	(*Valve 15, A+B*)
	(*Pin #1, 4, 8*)
		Valve15FB
			(
			Enable_Motion:= Enable_Motion,
			Enable_Latch:= TRUE,					(*Enabling Runs Valve as detent type (maintained solenoids*)
			Enable_SideA_PreCharge:= FALSE,		(*Enabling Turns Side A PreCharge Active, reset when Side B is energized in Auto*)
			Enable_SideB_PreCharge:= FALSE,		(*Enabling Turns Side B PreCharge Active, reset when Side A is energized in Auto*)
			PreCharge_Time:= T#0.10S,
			Enable_Auto_Commands:= In_Auto,
			Enable_Manual_Commands:= In_Manual AND (All_Robots_Clear OR TurntableB_At_Robot),  (*TLK ADDED OR*)
			In_Manual_SideA_Command:= (Discrete_In.ManReqs.28 OR Discrete_In.Go_Home),
			In_Manual_SideB_Command:= Discrete_In.ManReqs.29,
			SideA_Indicator:= (Pin1ADVD AND Pin4ADVD AND Pin8ADVD) OR Manual_Ind_HomePrompt,
			SideB_Indicator:= Pin1RETD AND Pin4RETD AND Pin8RETD,
			TurnOn_SideA_SOL=> N100.Q.28,
			TurnOn_SideB_SOL=> N100.Q.29,
			TurnOn_SideA_Indicator=> Manual_Indicators1.28,
			TurnOn_SideB_Indicator=> Manual_Indicators1.29
			 );
		Valve15FB.In_Auto_SideA_Command:= (Clamp_Step.0 AND NOT Unclamp_Step.0 OR Unclamp_Step.3)
										OR ((TurntableA_At_Robot OR Turntable_Bypassed) AND All_Sensors_Off AND Weld_Robots_Clear);
		Valve15FB.In_Auto_SideB_Command:= Unclamp_Step.0;


	(*Valve 16, A+B*)
	(*Clamp #5, 38, Slide #3, 5, 9, 12, 13*)
		Valve16FB
			(
			Enable_Motion:= Enable_Motion,
			Enable_Latch:= TRUE,					(*Enabling Runs Valve as detent type (maintained solenoids*)
			Enable_SideA_PreCharge:= FALSE,		(*Enabling Turns Side A PreCharge Active, reset when Side B is energized in Auto*)
			Enable_SideB_PreCharge:= FALSE,		(*Enabling Turns Side B PreCharge Active, reset when Side A is energized in Auto*)
			PreCharge_Time:= T#0.10S,
			Enable_Auto_Commands:= In_Auto,
			Enable_Manual_Commands:= In_Manual AND (All_Robots_Clear OR TurntableB_At_Robot),  (*TLK ADDED OR*)
			In_Manual_SideA_Command:= Discrete_In.ManReqs.30,
			In_Manual_SideB_Command:= (Discrete_In.ManReqs.31 OR Discrete_In.Go_Home),
			SideA_Indicator:= Clamp5ADVD AND Clamp38ADVD AND Slide3ADVD AND Slide5ADVD AND Slide9ADVD AND Slide12ADVD AND Slide13ADVD,
			SideB_Indicator:= (Clamp5RETD AND Clamp38RETD AND Slide3RETD AND Slide5RETD AND Slide9RETD AND Slide12RETD AND Slide13RETD) OR Manual_Ind_HomePrompt,
			TurnOn_SideA_SOL=> N100.Q.30,
			TurnOn_SideB_SOL=> N100.Q.31,
			TurnOn_SideA_Indicator=> Manual_Indicators1.30,
			TurnOn_SideB_Indicator=> Manual_Indicators1.31
			 );
		Valve16FB.In_Auto_SideA_Command:= (Clamp_Step.4 AND NOT Unclamp_Step.0);
		Valve16FB.In_Auto_SideB_Command:= Unclamp_Step.0
										OR ((TurntableA_At_Robot OR Turntable_Bypassed) AND All_Sensors_Off AND Weld_Robots_Clear);


























(*end*)
END_ACTION

ACTION ValveBank2:


(*+++++++++++THIS AREA IS CUSTOM PER INSTALLATION AND WILL HAVE TO BE MODIFIED PER +++++++++++++*)
(*+++++++++++THIS AREA IS CUSTOM PER INSTALLATION AND WILL HAVE TO BE MODIFIED PER +++++++++++++*)
(*+++++++++++THIS AREA IS CUSTOM PER INSTALLATION AND WILL HAVE TO BE MODIFIED PER +++++++++++++*)

(*+++++++++++VALVE BANK 2 +++++++++++++*)
(*+++++++++++VALVE BANK 2 +++++++++++++*)
(*+++++++++++VALVE BANK 2 +++++++++++++*)


	(*Valve 17, A+B*)
	(*QA Checks #1-6*)
		Valve17FB
			(
			Enable_Motion:= Enable_Motion ,
			Enable_Latch:= TRUE,					(*Enabling Runs Valve as detent type (maintained solenoids*)
			Enable_SideA_PreCharge:= FALSE,		(*Enabling Turns Side A PreCharge Active, reset when Side B is energized in Auto*)
			Enable_SideB_PreCharge:= FALSE,		(*Enabling Turns Side B PreCharge Active, reset when Side A is energized in Auto*)
			PreCharge_Time:= T#0.1S,
			Enable_Auto_Commands:= In_Auto,
			Enable_Manual_Commands:= In_Manual AND (All_Robots_Clear OR TurntableB_At_Robot),  (*TLK ADDED OR*)
			In_Manual_SideA_Command:= Discrete_In.ManReqs2.0,
			In_Manual_SideB_Command:= (Discrete_In.ManReqs2.1 OR Discrete_In.Go_Home),
			SideA_Indicator:= QACheck1ADVD AND QACheck2ADVD AND QACheck3ADVD AND QACheck4ADVD AND QACheck5ADVD AND QACheck6ADVD,
			SideB_Indicator:= (QACheck1RETD AND QACheck2RETD AND QACheck3RETD AND QACheck4RETD AND QACheck5RETD AND QACheck6RETD) OR Manual_Ind_HomePrompt,
			TurnOn_SideA_SOL=> N101.Q.0,
			TurnOn_SideB_SOL=> N101.Q.1,
			TurnOn_SideA_Indicator=> Manual_Indicators2.0,
			TurnOn_SideB_Indicator=> Manual_Indicators2.1
			 );
		Valve17FB.In_Auto_SideA_Command:= CheckQA1FB.Fire_QAchecks AND NOT Cycle_Complete;
		Valve17FB.In_Auto_SideB_Command:= NOT CheckQA1FB.Fire_QAchecks OR (Cycle_Complete AND All_Sensors_Off);


	(*Valve 18, ONLY 543*)
	(*Pin #3, 6*)
		Valve18FB
			(
			Enable_Motion:= Enable_Motion ,
			Enable_Latch:= FALSE,					(*Enabling Runs Valve as detent type (maintained solenoids*)
			Enable_SideA_PreCharge:= FALSE,		(*Enabling Turns Side A PreCharge Active, reset when Side B is energized in Auto*)
			Enable_SideB_PreCharge:= FALSE,		(*Enabling Turns Side B PreCharge Active, reset when Side A is energized in Auto*)
			PreCharge_Time:= T#0.10S,
			Enable_Auto_Commands:= In_Auto,
			Enable_Manual_Commands:= In_Manual AND (All_Robots_Clear OR TurntableB_At_Robot),  (*TLK ADDED OR*)
			In_Manual_SideA_Command:= Discrete_In.ManReqs2.2,
			In_Manual_SideB_Command:= (Discrete_In.ManReqs2.3 OR Discrete_In.Go_Home),
			SideA_Indicator:= Pin3ADVD AND Pin6ADVD,
			SideB_Indicator:= (Pin3RETD AND Pin6RETD) OR Manual_Ind_HomePrompt,
			TurnOn_SideA_SOL=> N101.Q.2,
			TurnOn_SideB_SOL=> N101.Q.3,
			TurnOn_SideA_Indicator=> Manual_Indicators2.2,
			TurnOn_SideB_Indicator=> Manual_Indicators2.3
			 );
	IF ((Model_ID=3) OR (Model_ID=10)) THEN		 
				Valve18FB.In_Auto_SideA_Command:= (Clamp_Step.2 AND NOT Unclamp_Step.0);
				Valve18FB.In_Auto_SideB_Command:= Unclamp_Step.0
												OR ((TurntableA_At_Robot OR Turntable_Bypassed) AND All_Sensors_Off AND Weld_Robots_Clear);
			ELSE
				Valve18FB.In_Auto_SideA_Command:= FALSE;
				Valve18FB.In_Auto_SideB_Command:= TRUE;
			END_IF
												
												
												
	(*Valve 19, ONLY 543*)
	(*Pin #2, 5, 7*)
		Valve19FB
			(
			Enable_Motion:= Enable_Motion,
			Enable_Latch:= FALSE,					(*Enabling Runs Valve as detent type (maintained solenoids*)
			Enable_SideA_PreCharge:= FALSE,		(*Enabling Turns Side A PreCharge Active, reset when Side B is energized in Auto*)
			Enable_SideB_PreCharge:= FALSE,		(*Enabling Turns Side B PreCharge Active, reset when Side A is energized in Auto*)
			PreCharge_Time:= T#0.10S,
			Enable_Auto_Commands:= In_Auto,
			Enable_Manual_Commands:= In_Manual AND (All_Robots_Clear OR TurntableB_At_Robot),  (*TLK ADDED OR*)
			In_Manual_SideA_Command:=  Discrete_In.ManReqs2.4 OR(Discrete_In.Go_Home AND Model_ID=3),
			In_Manual_SideB_Command:=  Discrete_In.ManReqs2.5 OR(Discrete_In.Go_Home AND Model_ID<>3),
			SideA_Indicator:= (Pin2ADVD AND Pin5ADVD AND Pin7ADVD) OR Manual_Ind_HomePrompt,
			SideB_Indicator:= (Pin2RETD AND Pin5RETD AND Pin7RETD) OR Manual_Ind_HomePrompt,
			TurnOn_SideA_SOL=> N101.Q.4,
			TurnOn_SideB_SOL=> N101.Q.5,
			TurnOn_SideA_Indicator=> Manual_Indicators2.4,
			TurnOn_SideB_Indicator=> Manual_Indicators2.5
			 );
	IF ((Model_ID=3) OR (Model_ID=10)) THEN		 
				Valve19FB.In_Auto_SideA_Command:= ((Clamp_Step.0 AND NOT Unclamp_Step.0))
												OR ((TurntableA_At_Robot OR Turntable_Bypassed) AND All_Sensors_Off AND Weld_Robots_Clear);
				Valve19FB.In_Auto_SideB_Command:= Unclamp_Step.0;
		ELSE
				Valve19FB.In_Auto_SideA_Command:= FALSE;
				Valve19FB.In_Auto_SideB_Command:= TRUE;
		END_IF
				
				

	(*Valve 20, ONLY 543*)
	(*Clamp #8, 24, 31*)
		Valve20FB
			(
			Enable_Motion:= Enable_Motion,
			Enable_Latch:= FALSE,					(*Enabling Runs Valve as detent type (maintained solenoids*)
			Enable_SideA_PreCharge:= FALSE,		(*Enabling Turns Side A PreCharge Active, reset when Side B is energized in Auto*)
			Enable_SideB_PreCharge:= FALSE,		(*Enabling Turns Side B PreCharge Active, reset when Side A is energized in Auto*)
			PreCharge_Time:= T#0.10S,
			Enable_Auto_Commands:= In_Auto,
			Enable_Manual_Commands:= In_Manual AND (All_Robots_Clear OR TurntableB_At_Robot),  (*TLK ADDED OR*)
			In_Manual_SideA_Command:= Discrete_In.ManReqs2.6,
			In_Manual_SideB_Command:= (Discrete_In.ManReqs2.7 OR Discrete_In.Go_Home),
			SideA_Indicator:= Clamp8ADVD AND Clamp24ADVD AND Clamp31ADVD,
			SideB_Indicator:= (Clamp8RETD AND Clamp24RETD AND Clamp31RETD) OR Manual_Ind_HomePrompt,
			TurnOn_SideA_SOL=> N101.Q.6,
			TurnOn_SideB_SOL=> N101.Q.7,
			TurnOn_SideA_Indicator=> Manual_Indicators2.6,
			TurnOn_SideB_Indicator=> Manual_Indicators2.7
			 );
			 
	IF ((Model_ID=3) OR (Model_ID=10)) THEN			 
				Valve20FB.In_Auto_SideA_Command:= (Clamp_Step.1 AND NOT Unclamp_Step.3);
				Valve20FB.In_Auto_SideB_Command:= Unclamp_Step.3
												OR ((TurntableA_At_Robot OR Turntable_Bypassed) AND All_Sensors_Off AND Weld_Robots_Clear);
		ELSE
				Valve20FB.In_Auto_SideA_Command:= FALSE;
				Valve20FB.In_Auto_SideB_Command:= TRUE;
		END_IF


	(*Valve 21, ONLY 543*)
	(*Clamp #10, 27*)
		Valve21FB
			(
			Enable_Motion:= Enable_Motion,
			Enable_Latch:= FALSE,					(*Enabling Runs Valve as detent type (maintained solenoids*)
			Enable_SideA_PreCharge:= FALSE,		(*Enabling Turns Side A PreCharge Active, reset when Side B is energized in Auto*)
			Enable_SideB_PreCharge:= FALSE,		(*Enabling Turns Side B PreCharge Active, reset when Side A is energized in Auto*)
			PreCharge_Time:= T#0.10S,
			Enable_Auto_Commands:= In_Auto,
			Enable_Manual_Commands:= In_Manual AND (All_Robots_Clear OR TurntableB_At_Robot),  (*TLK ADDED OR*)
			In_Manual_SideA_Command:= Discrete_In.ManReqs2.8,
			In_Manual_SideB_Command:= (Discrete_In.ManReqs2.9 OR Discrete_In.Go_Home),
			SideA_Indicator:= Clamp10ADVD AND Clamp27ADVD,
			SideB_Indicator:= (Clamp10RETD AND Clamp27RETD) OR Manual_Ind_HomePrompt,
			TurnOn_SideA_SOL=> N101.Q.8,
			TurnOn_SideB_SOL=> N101.Q.9,
			TurnOn_SideA_Indicator=> Manual_Indicators2.8,
			TurnOn_SideB_Indicator=> Manual_Indicators2.9
			 );
	IF ((Model_ID=3) OR (Model_ID=10)) THEN			 
				Valve21FB.In_Auto_SideA_Command:= (Clamp_Step.1 AND NOT Unclamp_Step.3);
				Valve21FB.In_Auto_SideB_Command:= Unclamp_Step.3
												OR ((TurntableA_At_Robot OR Turntable_Bypassed) AND All_Sensors_Off AND Weld_Robots_Clear);
		ELSE
				Valve21FB.In_Auto_SideA_Command:= FALSE;
				Valve21FB.In_Auto_SideB_Command:= TRUE;
		END_IF

	(*Valve 22, A+B*)
	(*LOCKS*)
		Valve22FB
			(
			Enable_Motion:= Enable_Motion ,
			Enable_Latch:= FALSE,					(*Enabling Runs Valve as detent type (maintained solenoids*)
			Enable_SideA_PreCharge:= FALSE,		(*Enabling Turns Side A PreCharge Active, reset when Side B is energized in Auto*)
			Enable_SideB_PreCharge:= FALSE,		(*Enabling Turns Side B PreCharge Active, reset when Side A is energized in Auto*)
			PreCharge_Time:= T#0.10S,
			Enable_Auto_Commands:= In_Auto,
			Enable_Manual_Commands:= In_Manual AND (All_Robots_Clear OR TurntableB_At_Robot),  (*TLK ADDED OR*)
			In_Manual_SideA_Command:= (Discrete_In.ManReqs2.10 OR Discrete_In.Go_Home)
										OR (N100.Q.18 AND NOT (Slide4ADVD AND Slide8ADVD AND Slide11ADVD))
										OR (N100.Q.19 AND NOT (Slide4RETD AND Slide8RETD AND Slide11RETD))
										OR (N100.Q.20 AND NOT (Slide6ADVD))
										OR (N100.Q.21 AND NOT (Slide6RETD))
										OR (N100.Q.22 AND NOT (Slide7ADVD))
										OR (N100.Q.23 AND NOT (Slide7RETD))
										OR (N100.Q.24 AND NOT (Slide10ADVD))
										OR (N100.Q.25 AND NOT (Slide10RETD))
										OR (N100.Q.26 AND NOT (Slide1ADVD AND Slide2ADVD AND Slide14ADVD AND Slide15ADVD))
										OR (N100.Q.27 AND NOT (Slide1RETD AND Slide2RETD AND Slide14RETD AND Slide15RETD))
										OR (N100.Q.30 AND NOT (Slide3ADVD AND Slide5ADVD AND Slide9ADVD AND Slide12ADVD AND Slide13ADVD))
										OR (N100.Q.31 AND NOT (Slide3RETD AND Slide5RETD AND Slide9RETD AND Slide12RETD AND Slide13RETD)),
			In_Manual_SideB_Command:= FALSE,
			SideA_Indicator:= Manual_Ind_HomePrompt,
			SideB_Indicator:= FALSE,
			TurnOn_SideA_SOL=> N101.Q.10,
			TurnOn_SideB_SOL=> N101.Q.11,
			TurnOn_SideA_Indicator=> Manual_Indicators2.10,
			TurnOn_SideB_Indicator=> Manual_Indicators2.11
			 );
		Valve22FB.In_Auto_SideA_Command:= (N100.Q.18 AND NOT (Slide4ADVD AND Slide8ADVD AND Slide11ADVD))
										OR (N100.Q.19 AND NOT (Slide4RETD AND Slide8RETD AND Slide11RETD))
										OR (N100.Q.20 AND NOT (Slide6ADVD))
										OR (N100.Q.21 AND NOT (Slide6RETD))
										OR (N100.Q.22 AND NOT (Slide7ADVD))
										OR (N100.Q.23 AND NOT (Slide7RETD))
										OR (N100.Q.24 AND NOT (Slide10ADVD))
										OR (N100.Q.25 AND NOT (Slide10RETD))
										OR (N100.Q.26 AND NOT (Slide1ADVD AND Slide2ADVD AND Slide14ADVD AND Slide15ADVD))
										OR (N100.Q.27 AND NOT (Slide1RETD AND Slide2RETD AND Slide14RETD AND Slide15RETD))
										OR (N100.Q.30 AND NOT (Slide3ADVD AND Slide5ADVD AND Slide9ADVD AND Slide12ADVD AND Slide13ADVD))
										OR (N100.Q.31 AND NOT (Slide3RETD AND Slide5RETD AND Slide9RETD AND Slide12RETD AND Slide13RETD));
		Valve22FB.In_Auto_SideB_Command:= FALSE;

	(*Valve 23, A+B*)
	(*Spare*)
		Valve23FB
			(
			Enable_Motion:= Enable_Motion,
			Enable_Latch:= FALSE,					(*Enabling Runs Valve as detent type (maintained solenoids*)
			Enable_SideA_PreCharge:= FALSE,		(*Enabling Turns Side A PreCharge Active, reset when Side B is energized in Auto*)
			Enable_SideB_PreCharge:= FALSE,		(*Enabling Turns Side B PreCharge Active, reset when Side A is energized in Auto*)
			PreCharge_Time:= T#0.10S,
			Enable_Auto_Commands:= In_Auto,
			Enable_Manual_Commands:= In_Manual AND (All_Robots_Clear OR TurntableB_At_Robot),  (*TLK ADDED OR*)
			In_Manual_SideA_Command:= Discrete_In.ManReqs2.12,
			In_Manual_SideB_Command:= Discrete_In.ManReqs2.13 OR Discrete_In.Go_Home,
			SideA_Indicator:= (*Clamp21ADVD*) FALSE,
			SideB_Indicator:= (*Clamp21RETD*) FALSE,
			TurnOn_SideA_SOL=> N101.Q.12,
			TurnOn_SideB_SOL=> N101.Q.13,
			TurnOn_SideA_Indicator=> Manual_Indicators2.12,
			TurnOn_SideB_Indicator=> Manual_Indicators2.13
			 );
		Valve23FB.In_Auto_SideA_Command:= (*Clamp_Step.1 AND NOT Unclamp_Step.0*) FALSE;
		Valve23FB.In_Auto_SideB_Command:= (*Unclamp_Step.0
										OR ((TurntableA_At_Robot OR Turntable_Bypassed) AND All_Sensors_Off AND Weld_Robots_Clear)*) FALSE;


(*---------------------------------------------------------SPARE---------------------------------------------------------*)		


	(*Valve 24, A+B*)
	(*spare*)
		Valve24FB
			(
			Enable_Motion:= Enable_Motion ,
			Enable_Latch:= TRUE,					(*Enabling Runs Valve as detent type (maintained solenoids*)
			Enable_SideA_PreCharge:= FALSE,		(*Enabling Turns Side A PreCharge Active, reset when Side B is energized in Auto*)
			Enable_SideB_PreCharge:= FALSE,		(*Enabling Turns Side B PreCharge Active, reset when Side A is energized in Auto*)
			PreCharge_Time:= T#0.10S,
			Enable_Auto_Commands:= In_Auto,
			Enable_Manual_Commands:= In_Manual AND (All_Robots_Clear OR TurntableB_At_Robot),  (*TLK ADDED OR*)
			In_Manual_SideA_Command:= Discrete_In.ManReqs2.14,
			In_Manual_SideB_Command:= Discrete_In.ManReqs2.15,
			SideA_Indicator:= FALSE,
			SideB_Indicator:= FALSE,
			TurnOn_SideA_SOL=> N101.Q.14,
			TurnOn_SideB_SOL=> N101.Q.15,
			TurnOn_SideA_Indicator=> Manual_Indicators2.14,
			TurnOn_SideB_Indicator=> Manual_Indicators2.15
			 );
		Valve24FB.In_Auto_SideA_Command:= FALSE;
		Valve24FB.In_Auto_SideB_Command:= FALSE;


	(*Valve 25, A+B*)
	(*spare*)
		Valve25FB
			(
			Enable_Motion:= Enable_Motion ,
			Enable_Latch:= TRUE,					(*Enabling Runs Valve as detent type (maintained solenoids*)
			Enable_SideA_PreCharge:= FALSE,		(*Enabling Turns Side A PreCharge Active, reset when Side B is energized in Auto*)
			Enable_SideB_PreCharge:= FALSE,		(*Enabling Turns Side B PreCharge Active, reset when Side A is energized in Auto*)
			PreCharge_Time:= T#0.10S,
			Enable_Auto_Commands:= In_Auto,
			Enable_Manual_Commands:= In_Manual AND (All_Robots_Clear OR TurntableB_At_Robot),  (*TLK ADDED OR*)
			In_Manual_SideA_Command:= Discrete_In.ManReqs2.16,
			In_Manual_SideB_Command:= Discrete_In.ManReqs2.17,
			SideA_Indicator:= FALSE,
			SideB_Indicator:= FALSE,
			TurnOn_SideA_SOL=> N101.Q.16,
			TurnOn_SideB_SOL=> N101.Q.17,
			TurnOn_SideA_Indicator=> Manual_Indicators2.16,
			TurnOn_SideB_Indicator=> Manual_Indicators2.17
			 );
		Valve25FB.In_Auto_SideA_Command:= FALSE;
		Valve25FB.In_Auto_SideB_Command:= FALSE;


	(*Valve 26, A+B*)
	(*spare*)
		Valve26FB
			(
			Enable_Motion:= Enable_Motion ,
			Enable_Latch:= TRUE,					(*Enabling Runs Valve as detent type (maintained solenoids*)
			Enable_SideA_PreCharge:= FALSE,		(*Enabling Turns Side A PreCharge Active, reset when Side B is energized in Auto*)
			Enable_SideB_PreCharge:= FALSE,		(*Enabling Turns Side B PreCharge Active, reset when Side A is energized in Auto*)
			PreCharge_Time:= T#0.10S,
			Enable_Auto_Commands:= In_Auto,
			Enable_Manual_Commands:= In_Manual AND (All_Robots_Clear OR TurntableB_At_Robot),  (*TLK ADDED OR*)
			In_Manual_SideA_Command:= Discrete_In.ManReqs2.18,
			In_Manual_SideB_Command:= Discrete_In.ManReqs2.19,
			SideA_Indicator:= FALSE,
			SideB_Indicator:= FALSE,
			TurnOn_SideA_SOL=> N101.Q.18,
			TurnOn_SideB_SOL=> N101.Q.19,
			TurnOn_SideA_Indicator=> Manual_Indicators2.18,
			TurnOn_SideB_Indicator=> Manual_Indicators2.19
			 );
		Valve26FB.In_Auto_SideA_Command:= FALSE;
		Valve26FB.In_Auto_SideB_Command:= FALSE;


	(*Valve 27, A+B*)
	(*spare*)
		Valve27FB
			(
			Enable_Motion:= Enable_Motion ,
			Enable_Latch:= TRUE,					(*Enabling Runs Valve as detent type (maintained solenoids*)
			Enable_SideA_PreCharge:= FALSE,		(*Enabling Turns Side A PreCharge Active, reset when Side B is energized in Auto*)
			Enable_SideB_PreCharge:= FALSE,		(*Enabling Turns Side B PreCharge Active, reset when Side A is energized in Auto*)
			PreCharge_Time:= T#0.10S,
			Enable_Auto_Commands:= In_Auto,
			Enable_Manual_Commands:= In_Manual AND (All_Robots_Clear OR TurntableB_At_Robot),  (*TLK ADDED OR*)
			In_Manual_SideA_Command:= Discrete_In.ManReqs2.20,
			In_Manual_SideB_Command:= Discrete_In.ManReqs2.21,
			SideA_Indicator:= FALSE,
			SideB_Indicator:= FALSE,
			TurnOn_SideA_SOL=> N101.Q.20,
			TurnOn_SideB_SOL=> N101.Q.21,
			TurnOn_SideA_Indicator=> Manual_Indicators2.20,
			TurnOn_SideB_Indicator=> Manual_Indicators2.21
			 );
		Valve27FB.In_Auto_SideA_Command:= FALSE;
		Valve27FB.In_Auto_SideB_Command:= FALSE;


	(*Valve 28, A+B*)
	(*spare*)
		Valve28FB
			(
			Enable_Motion:= Enable_Motion ,
			Enable_Latch:= TRUE,					(*Enabling Runs Valve as detent type (maintained solenoids*)
			Enable_SideA_PreCharge:= FALSE,		(*Enabling Turns Side A PreCharge Active, reset when Side B is energized in Auto*)
			Enable_SideB_PreCharge:= FALSE,		(*Enabling Turns Side B PreCharge Active, reset when Side A is energized in Auto*)
			PreCharge_Time:= T#0.10S,
			Enable_Auto_Commands:= In_Auto,
			Enable_Manual_Commands:= In_Manual AND (All_Robots_Clear OR TurntableB_At_Robot),  (*TLK ADDED OR*)
			In_Manual_SideA_Command:= Discrete_In.ManReqs2.22,
			In_Manual_SideB_Command:= Discrete_In.ManReqs2.23,
			SideA_Indicator:= FALSE,
			SideB_Indicator:= FALSE,
			TurnOn_SideA_SOL=> N101.Q.22,
			TurnOn_SideB_SOL=> N101.Q.23,
			TurnOn_SideA_Indicator=> Manual_Indicators2.22,
			TurnOn_SideB_Indicator=> Manual_Indicators2.23
			 );
		Valve28FB.In_Auto_SideA_Command:= FALSE;
		Valve28FB.In_Auto_SideB_Command:= FALSE;


	(*Valve 29, A+B*)
	(*spare*)
		Valve29FB
			(
			Enable_Motion:= Enable_Motion ,
			Enable_Latch:= TRUE,					(*Enabling Runs Valve as detent type (maintained solenoids*)
			Enable_SideA_PreCharge:= FALSE,		(*Enabling Turns Side A PreCharge Active, reset when Side B is energized in Auto*)
			Enable_SideB_PreCharge:= FALSE,		(*Enabling Turns Side B PreCharge Active, reset when Side A is energized in Auto*)
			PreCharge_Time:= T#0.10S,
			Enable_Auto_Commands:= In_Auto,
			Enable_Manual_Commands:= In_Manual AND (All_Robots_Clear OR TurntableB_At_Robot),  (*TLK ADDED OR*)
			In_Manual_SideA_Command:= Discrete_In.ManReqs2.24,
			In_Manual_SideB_Command:= Discrete_In.ManReqs2.25,
			SideA_Indicator:= FALSE,
			SideB_Indicator:= FALSE,
			TurnOn_SideA_SOL=> N101.Q.24,
			TurnOn_SideB_SOL=> N101.Q.25,
			TurnOn_SideA_Indicator=> Manual_Indicators2.24,
			TurnOn_SideB_Indicator=> Manual_Indicators2.25
			 );
		Valve29FB.In_Auto_SideA_Command:= FALSE;
		Valve29FB.In_Auto_SideB_Command:= FALSE;


	(*Valve 30, A+B*)
	(*spare*)
		Valve30FB
			(
			Enable_Motion:= Enable_Motion ,
			Enable_Latch:= TRUE,					(*Enabling Runs Valve as detent type (maintained solenoids*)
			Enable_SideA_PreCharge:= FALSE,		(*Enabling Turns Side A PreCharge Active, reset when Side B is energized in Auto*)
			Enable_SideB_PreCharge:= FALSE,		(*Enabling Turns Side B PreCharge Active, reset when Side A is energized in Auto*)
			PreCharge_Time:= T#0.10S,
			Enable_Auto_Commands:= In_Auto,
			Enable_Manual_Commands:= In_Manual AND (All_Robots_Clear OR TurntableB_At_Robot),  (*TLK ADDED OR*)
			In_Manual_SideA_Command:= Discrete_In.ManReqs2.26,
			In_Manual_SideB_Command:= Discrete_In.ManReqs2.27,
			SideA_Indicator:= FALSE,
			SideB_Indicator:= FALSE,
			TurnOn_SideA_SOL=> N101.Q.26,
			TurnOn_SideB_SOL=> N101.Q.27,
			TurnOn_SideA_Indicator=> Manual_Indicators2.26,
			TurnOn_SideB_Indicator=> Manual_Indicators2.27
			 );
		Valve30FB.In_Auto_SideA_Command:= FALSE;
		Valve30FB.In_Auto_SideB_Command:= FALSE;


	(*Valve 31, A+B*)
	(*spare*)
		Valve31FB
			(
			Enable_Motion:= Enable_Motion ,
			Enable_Latch:= TRUE,					(*Enabling Runs Valve as detent type (maintained solenoids*)
			Enable_SideA_PreCharge:= FALSE,		(*Enabling Turns Side A PreCharge Active, reset when Side B is energized in Auto*)
			Enable_SideB_PreCharge:= FALSE,		(*Enabling Turns Side B PreCharge Active, reset when Side A is energized in Auto*)
			PreCharge_Time:= T#0.10S,
			Enable_Auto_Commands:= In_Auto,
			Enable_Manual_Commands:= In_Manual AND (All_Robots_Clear OR TurntableB_At_Robot),  (*TLK ADDED OR*)
			In_Manual_SideA_Command:= Discrete_In.ManReqs2.28,
			In_Manual_SideB_Command:= Discrete_In.ManReqs2.29,
			SideA_Indicator:= FALSE,
			SideB_Indicator:= FALSE,
			TurnOn_SideA_SOL=> N101.Q.28,
			TurnOn_SideB_SOL=> N101.Q.29,
			TurnOn_SideA_Indicator=> Manual_Indicators2.28,
			TurnOn_SideB_Indicator=> Manual_Indicators2.29
			 );
		Valve31FB.In_Auto_SideA_Command:= FALSE;
		Valve31FB.In_Auto_SideB_Command:= FALSE;


	(*Valve 32, A+B*)
	(*spare*)
		Valve32FB
			(
			Enable_Motion:= Enable_Motion ,
			Enable_Latch:= TRUE,					(*Enabling Runs Valve as detent type (maintained solenoids*)
			Enable_SideA_PreCharge:= FALSE,		(*Enabling Turns Side A PreCharge Active, reset when Side B is energized in Auto*)
			Enable_SideB_PreCharge:= FALSE,		(*Enabling Turns Side B PreCharge Active, reset when Side A is energized in Auto*)
			PreCharge_Time:= T#0.10S,
			Enable_Auto_Commands:= In_Auto,
			Enable_Manual_Commands:= In_Manual AND (All_Robots_Clear OR TurntableB_At_Robot),  (*TLK ADDED OR*)
			In_Manual_SideA_Command:= Discrete_In.ManReqs2.30,
			In_Manual_SideB_Command:= Discrete_In.ManReqs2.31,
			SideA_Indicator:= FALSE,
			SideB_Indicator:= FALSE,
			TurnOn_SideA_SOL=> N101.Q.30,
			TurnOn_SideB_SOL=> N101.Q.31,
			TurnOn_SideA_Indicator=> Manual_Indicators2.30,
			TurnOn_SideB_Indicator=> Manual_Indicators2.31
			 );
		Valve32FB.In_Auto_SideA_Command:= FALSE;
		Valve32FB.In_Auto_SideB_Command:= FALSE;




















(*end*)
END_ACTION

ACTION ValveBank3:


(*+++++++++++THIS AREA IS CUSTOM PER INSTALLATION AND WILL HAVE TO BE MODIFIED PER +++++++++++++*)
(*+++++++++++THIS AREA IS CUSTOM PER INSTALLATION AND WILL HAVE TO BE MODIFIED PER +++++++++++++*)
(*+++++++++++THIS AREA IS CUSTOM PER INSTALLATION AND WILL HAVE TO BE MODIFIED PER +++++++++++++*)

(*+++++++++++VALVE BANK 3 +++++++++++++*)
(*+++++++++++VALVE BANK 3 +++++++++++++*)
(*+++++++++++VALVE BANK 3 +++++++++++++*)


	(*Valve 33, A+B*)
	(*spare*)
		Valve33FB
			(
			Enable_Motion:= Enable_Motion ,
			Enable_Latch:= TRUE,					(*Enabling Runs Valve as detent type (maintained solenoids*)
			Enable_SideA_PreCharge:= FALSE,		(*Enabling Turns Side A PreCharge Active, reset when Side B is energized in Auto*)
			Enable_SideB_PreCharge:= FALSE,		(*Enabling Turns Side B PreCharge Active, reset when Side A is energized in Auto*)
			PreCharge_Time:= T#0.1S,
			Enable_Auto_Commands:= In_Auto,
			Enable_Manual_Commands:= In_Manual AND All_Robots_Clear,
			In_Manual_SideA_Command:= Discrete_In.ManReqs3.0,
			In_Manual_SideB_Command:= (Discrete_In.ManReqs3.1 OR Discrete_In.Go_Home),
			SideA_Indicator:= FALSE,
			SideB_Indicator:= FALSE,
			TurnOn_SideA_SOL=> N102.Q.0,
			TurnOn_SideB_SOL=> N102.Q.1,
			TurnOn_SideA_Indicator=> Manual_Indicators3.0,
			TurnOn_SideB_Indicator=> Manual_Indicators3.1
			 );
		Valve33FB.In_Auto_SideA_Command:= FALSE;
		Valve33FB.In_Auto_SideB_Command:= FALSE;


	(*Valve 34, A+B*)
	(*spare*)
		Valve34FB
			(
			Enable_Motion:= Enable_Motion ,
			Enable_Latch:= TRUE,					(*Enabling Runs Valve as detent type (maintained solenoids*)
			Enable_SideA_PreCharge:= FALSE,		(*Enabling Turns Side A PreCharge Active, reset when Side B is energized in Auto*)
			Enable_SideB_PreCharge:= FALSE,		(*Enabling Turns Side B PreCharge Active, reset when Side A is energized in Auto*)
			PreCharge_Time:= T#0.10S,
			Enable_Auto_Commands:= In_Auto,
			Enable_Manual_Commands:= In_Manual AND All_Robots_Clear,
			In_Manual_SideA_Command:= Discrete_In.ManReqs3.2,
			In_Manual_SideB_Command:= Discrete_In.ManReqs3.3,
			SideA_Indicator:= FALSE,
			SideB_Indicator:= FALSE,
			TurnOn_SideA_SOL=> N102.Q.2,
			TurnOn_SideB_SOL=> N102.Q.3,
			TurnOn_SideA_Indicator=> Manual_Indicators3.2,
			TurnOn_SideB_Indicator=> Manual_Indicators3.3
			 );
		Valve34FB.In_Auto_SideA_Command:= FALSE;
		Valve34FB.In_Auto_SideB_Command:= FALSE;


	(*Valve 35, A+B*)
	(*spare*)
		Valve35FB
			(
			Enable_Motion:= Enable_Motion ,
			Enable_Latch:= TRUE,					(*Enabling Runs Valve as detent type (maintained solenoids*)
			Enable_SideA_PreCharge:= FALSE,		(*Enabling Turns Side A PreCharge Active, reset when Side B is energized in Auto*)
			Enable_SideB_PreCharge:= FALSE,		(*Enabling Turns Side B PreCharge Active, reset when Side A is energized in Auto*)
			PreCharge_Time:= T#0.10S,
			Enable_Auto_Commands:= In_Auto,
			Enable_Manual_Commands:= In_Manual AND All_Robots_Clear,
			In_Manual_SideA_Command:= Discrete_In.ManReqs3.4,
			In_Manual_SideB_Command:= Discrete_In.ManReqs3.5,
			SideA_Indicator:= FALSE,
			SideB_Indicator:= FALSE,
			TurnOn_SideA_SOL=> N102.Q.4,
			TurnOn_SideB_SOL=> N102.Q.5,
			TurnOn_SideA_Indicator=> Manual_Indicators3.4,
			TurnOn_SideB_Indicator=> Manual_Indicators3.5
			 );
		Valve35FB.In_Auto_SideA_Command:= FALSE;
		Valve35FB.In_Auto_SideB_Command:= FALSE;


	(*Valve 36, A+B*)
	(*spare*)
		Valve36FB
			(
			Enable_Motion:= Enable_Motion ,
			Enable_Latch:= TRUE,					(*Enabling Runs Valve as detent type (maintained solenoids*)
			Enable_SideA_PreCharge:= FALSE,		(*Enabling Turns Side A PreCharge Active, reset when Side B is energized in Auto*)
			Enable_SideB_PreCharge:= FALSE,		(*Enabling Turns Side B PreCharge Active, reset when Side A is energized in Auto*)
			PreCharge_Time:= T#0.10S,
			Enable_Auto_Commands:= In_Auto,
			Enable_Manual_Commands:= In_Manual AND All_Robots_Clear,
			In_Manual_SideA_Command:= Discrete_In.ManReqs3.6,
			In_Manual_SideB_Command:= Discrete_In.ManReqs3.7,
			SideA_Indicator:= FALSE,
			SideB_Indicator:= FALSE,
			TurnOn_SideA_SOL=> N102.Q.6,
			TurnOn_SideB_SOL=> N102.Q.7,
			TurnOn_SideA_Indicator=> Manual_Indicators3.6,
			TurnOn_SideB_Indicator=> Manual_Indicators3.7
			 );
		Valve36FB.In_Auto_SideA_Command:= FALSE;
		Valve36FB.In_Auto_SideB_Command:= FALSE;


	(*Valve 37, A+B*)
	(*spare*)
		Valve37FB
			(
			Enable_Motion:= Enable_Motion ,
			Enable_Latch:= TRUE,					(*Enabling Runs Valve as detent type (maintained solenoids*)
			Enable_SideA_PreCharge:= FALSE,		(*Enabling Turns Side A PreCharge Active, reset when Side B is energized in Auto*)
			Enable_SideB_PreCharge:= FALSE,		(*Enabling Turns Side B PreCharge Active, reset when Side A is energized in Auto*)
			PreCharge_Time:= T#0.10S,
			Enable_Auto_Commands:= In_Auto,
			Enable_Manual_Commands:= In_Manual AND All_Robots_Clear,
			In_Manual_SideA_Command:= Discrete_In.ManReqs3.8,
			In_Manual_SideB_Command:= Discrete_In.ManReqs3.9,
			SideA_Indicator:= FALSE,
			SideB_Indicator:= FALSE,
			TurnOn_SideA_SOL=> N102.Q.8,
			TurnOn_SideB_SOL=> N102.Q.9,
			TurnOn_SideA_Indicator=> Manual_Indicators3.8,
			TurnOn_SideB_Indicator=> Manual_Indicators3.9
			 );
		Valve37FB.In_Auto_SideA_Command:= FALSE;
		Valve37FB.In_Auto_SideB_Command:= FALSE;


	(*Valve 38, A+B*)
	(*spare*)
		Valve38FB
			(
			Enable_Motion:= Enable_Motion ,
			Enable_Latch:= TRUE,					(*Enabling Runs Valve as detent type (maintained solenoids*)
			Enable_SideA_PreCharge:= FALSE,		(*Enabling Turns Side A PreCharge Active, reset when Side B is energized in Auto*)
			Enable_SideB_PreCharge:= FALSE,		(*Enabling Turns Side B PreCharge Active, reset when Side A is energized in Auto*)
			PreCharge_Time:= T#0.10S,
			Enable_Auto_Commands:= In_Auto,
			Enable_Manual_Commands:= In_Manual AND All_Robots_Clear,
			In_Manual_SideA_Command:= Discrete_In.ManReqs3.10,
			In_Manual_SideB_Command:= Discrete_In.ManReqs3.11,
			SideA_Indicator:= FALSE,
			SideB_Indicator:= FALSE,
			TurnOn_SideA_SOL=> N102.Q.10,
			TurnOn_SideB_SOL=> N102.Q.11,
			TurnOn_SideA_Indicator=> Manual_Indicators3.10,
			TurnOn_SideB_Indicator=> Manual_Indicators3.11
			 );
		Valve38FB.In_Auto_SideA_Command:= FALSE;
		Valve38FB.In_Auto_SideB_Command:= FALSE;


	(*Valve 39, A+B*)
	(*spare*)
		Valve39FB
			(
			Enable_Motion:= Enable_Motion ,
			Enable_Latch:= TRUE,					(*Enabling Runs Valve as detent type (maintained solenoids*)
			Enable_SideA_PreCharge:= FALSE,		(*Enabling Turns Side A PreCharge Active, reset when Side B is energized in Auto*)
			Enable_SideB_PreCharge:= FALSE,		(*Enabling Turns Side B PreCharge Active, reset when Side A is energized in Auto*)
			PreCharge_Time:= T#0.10S,
			Enable_Auto_Commands:= In_Auto,
			Enable_Manual_Commands:= In_Manual AND All_Robots_Clear,
			In_Manual_SideA_Command:= Discrete_In.ManReqs3.12,
			In_Manual_SideB_Command:= Discrete_In.ManReqs3.13,
			SideA_Indicator:= FALSE,
			SideB_Indicator:= FALSE,
			TurnOn_SideA_SOL=> N102.Q.12,
			TurnOn_SideB_SOL=> N102.Q.13,
			TurnOn_SideA_Indicator=> Manual_Indicators3.12,
			TurnOn_SideB_Indicator=> Manual_Indicators3.13
			 );
		Valve39FB.In_Auto_SideA_Command:= FALSE;
		Valve39FB.In_Auto_SideB_Command:= FALSE;


	(*Valve 40, A+B*)
	(*spare*)
		Valve40FB
			(
			Enable_Motion:= Enable_Motion ,
			Enable_Latch:= TRUE,					(*Enabling Runs Valve as detent type (maintained solenoids*)
			Enable_SideA_PreCharge:= FALSE,		(*Enabling Turns Side A PreCharge Active, reset when Side B is energized in Auto*)
			Enable_SideB_PreCharge:= FALSE,		(*Enabling Turns Side B PreCharge Active, reset when Side A is energized in Auto*)
			PreCharge_Time:= T#0.10S,
			Enable_Auto_Commands:= In_Auto,
			Enable_Manual_Commands:= In_Manual AND All_Robots_Clear,
			In_Manual_SideA_Command:= Discrete_In.ManReqs3.14,
			In_Manual_SideB_Command:= Discrete_In.ManReqs3.15,
			SideA_Indicator:= FALSE,
			SideB_Indicator:= FALSE,
			TurnOn_SideA_SOL=> N102.Q.14,
			TurnOn_SideB_SOL=> N102.Q.15,
			TurnOn_SideA_Indicator=> Manual_Indicators3.14,
			TurnOn_SideB_Indicator=> Manual_Indicators3.15
			 );
		Valve40FB.In_Auto_SideA_Command:= FALSE;
		Valve40FB.In_Auto_SideB_Command:= FALSE;


	(*Valve 41, A+B*)
	(*spare*)
		Valve41FB
			(
			Enable_Motion:= Enable_Motion ,
			Enable_Latch:= TRUE,					(*Enabling Runs Valve as detent type (maintained solenoids*)
			Enable_SideA_PreCharge:= FALSE,		(*Enabling Turns Side A PreCharge Active, reset when Side B is energized in Auto*)
			Enable_SideB_PreCharge:= FALSE,		(*Enabling Turns Side B PreCharge Active, reset when Side A is energized in Auto*)
			PreCharge_Time:= T#0.10S,
			Enable_Auto_Commands:= In_Auto,
			Enable_Manual_Commands:= In_Manual AND All_Robots_Clear,
			In_Manual_SideA_Command:= Discrete_In.ManReqs3.16,
			In_Manual_SideB_Command:= Discrete_In.ManReqs3.17,
			SideA_Indicator:= FALSE,
			SideB_Indicator:= FALSE,
			TurnOn_SideA_SOL=> N102.Q.16,
			TurnOn_SideB_SOL=> N102.Q.17,
			TurnOn_SideA_Indicator=> Manual_Indicators3.16,
			TurnOn_SideB_Indicator=> Manual_Indicators3.17
			 );
		Valve41FB.In_Auto_SideA_Command:= FALSE;
		Valve41FB.In_Auto_SideB_Command:= FALSE;


	(*Valve 42, A+B*)
	(*spare*)
		Valve42FB
			(
			Enable_Motion:= Enable_Motion ,
			Enable_Latch:= TRUE,					(*Enabling Runs Valve as detent type (maintained solenoids*)
			Enable_SideA_PreCharge:= FALSE,		(*Enabling Turns Side A PreCharge Active, reset when Side B is energized in Auto*)
			Enable_SideB_PreCharge:= FALSE,		(*Enabling Turns Side B PreCharge Active, reset when Side A is energized in Auto*)
			PreCharge_Time:= T#0.10S,
			Enable_Auto_Commands:= In_Auto,
			Enable_Manual_Commands:= In_Manual AND All_Robots_Clear,
			In_Manual_SideA_Command:= Discrete_In.ManReqs3.18,
			In_Manual_SideB_Command:= Discrete_In.ManReqs3.19,
			SideA_Indicator:= FALSE,
			SideB_Indicator:= FALSE,
			TurnOn_SideA_SOL=> N102.Q.18,
			TurnOn_SideB_SOL=> N102.Q.19,
			TurnOn_SideA_Indicator=> Manual_Indicators3.18,
			TurnOn_SideB_Indicator=> Manual_Indicators3.19
			 );
		Valve42FB.In_Auto_SideA_Command:= FALSE;
		Valve42FB.In_Auto_SideB_Command:= FALSE;


	(*Valve 43, A+B*)
	(*spare*)
		Valve43FB
			(
			Enable_Motion:= Enable_Motion ,
			Enable_Latch:= TRUE,					(*Enabling Runs Valve as detent type (maintained solenoids*)
			Enable_SideA_PreCharge:= FALSE,		(*Enabling Turns Side A PreCharge Active, reset when Side B is energized in Auto*)
			Enable_SideB_PreCharge:= FALSE,		(*Enabling Turns Side B PreCharge Active, reset when Side A is energized in Auto*)
			PreCharge_Time:= T#0.10S,
			Enable_Auto_Commands:= In_Auto,
			Enable_Manual_Commands:= In_Manual AND All_Robots_Clear,
			In_Manual_SideA_Command:= Discrete_In.ManReqs3.20,
			In_Manual_SideB_Command:= Discrete_In.ManReqs3.21,
			SideA_Indicator:= FALSE,
			SideB_Indicator:= FALSE,
			TurnOn_SideA_SOL=> N102.Q.20,
			TurnOn_SideB_SOL=> N102.Q.21,
			TurnOn_SideA_Indicator=> Manual_Indicators3.20,
			TurnOn_SideB_Indicator=> Manual_Indicators3.21
			 );
		Valve43FB.In_Auto_SideA_Command:= FALSE;
		Valve43FB.In_Auto_SideB_Command:= FALSE;


	(*Valve 44, A+B*)
	(*spare*)
		Valve44FB
			(
			Enable_Motion:= Enable_Motion ,
			Enable_Latch:= TRUE,					(*Enabling Runs Valve as detent type (maintained solenoids*)
			Enable_SideA_PreCharge:= FALSE,		(*Enabling Turns Side A PreCharge Active, reset when Side B is energized in Auto*)
			Enable_SideB_PreCharge:= FALSE,		(*Enabling Turns Side B PreCharge Active, reset when Side A is energized in Auto*)
			PreCharge_Time:= T#0.10S,
			Enable_Auto_Commands:= In_Auto,
			Enable_Manual_Commands:= In_Manual AND All_Robots_Clear,
			In_Manual_SideA_Command:= Discrete_In.ManReqs3.22,
			In_Manual_SideB_Command:= Discrete_In.ManReqs3.23,
			SideA_Indicator:= FALSE,
			SideB_Indicator:= FALSE,
			TurnOn_SideA_SOL=> N102.Q.22,
			TurnOn_SideB_SOL=> N102.Q.23,
			TurnOn_SideA_Indicator=> Manual_Indicators3.22,
			TurnOn_SideB_Indicator=> Manual_Indicators3.23
			 );
		Valve44FB.In_Auto_SideA_Command:= FALSE;
		Valve44FB.In_Auto_SideB_Command:= FALSE;


	(*Valve 45, A+B*)
	(*spare*)
		Valve45FB
			(
			Enable_Motion:= Enable_Motion ,
			Enable_Latch:= TRUE,					(*Enabling Runs Valve as detent type (maintained solenoids*)
			Enable_SideA_PreCharge:= FALSE,		(*Enabling Turns Side A PreCharge Active, reset when Side B is energized in Auto*)
			Enable_SideB_PreCharge:= FALSE,		(*Enabling Turns Side B PreCharge Active, reset when Side A is energized in Auto*)
			PreCharge_Time:= T#0.10S,
			Enable_Auto_Commands:= In_Auto,
			Enable_Manual_Commands:= In_Manual AND All_Robots_Clear,
			In_Manual_SideA_Command:= Discrete_In.ManReqs3.24,
			In_Manual_SideB_Command:= Discrete_In.ManReqs3.25,
			SideA_Indicator:= FALSE,
			SideB_Indicator:= FALSE,
			TurnOn_SideA_SOL=> N102.Q.24,
			TurnOn_SideB_SOL=> N102.Q.25,
			TurnOn_SideA_Indicator=> Manual_Indicators3.24,
			TurnOn_SideB_Indicator=> Manual_Indicators3.25
			 );
		Valve45FB.In_Auto_SideA_Command:= FALSE;
		Valve45FB.In_Auto_SideB_Command:= FALSE;


	(*Valve 46, A+B*)
	(*spare*)
		Valve46FB
			(
			Enable_Motion:= Enable_Motion ,
			Enable_Latch:= TRUE,					(*Enabling Runs Valve as detent type (maintained solenoids*)
			Enable_SideA_PreCharge:= FALSE,		(*Enabling Turns Side A PreCharge Active, reset when Side B is energized in Auto*)
			Enable_SideB_PreCharge:= FALSE,		(*Enabling Turns Side B PreCharge Active, reset when Side A is energized in Auto*)
			PreCharge_Time:= T#0.10S,
			Enable_Auto_Commands:= In_Auto,
			Enable_Manual_Commands:= In_Manual AND All_Robots_Clear,
			In_Manual_SideA_Command:= Discrete_In.ManReqs3.26,
			In_Manual_SideB_Command:= Discrete_In.ManReqs3.27,
			SideA_Indicator:= FALSE,
			SideB_Indicator:= FALSE,
			TurnOn_SideA_SOL=> N102.Q.26,
			TurnOn_SideB_SOL=> N102.Q.27,
			TurnOn_SideA_Indicator=> Manual_Indicators3.26,
			TurnOn_SideB_Indicator=> Manual_Indicators3.27
			 );
		Valve46FB.In_Auto_SideA_Command:= FALSE;
		Valve46FB.In_Auto_SideB_Command:= FALSE;


	(*Valve 47, A+B*)
	(*spare*)
		Valve47FB
			(
			Enable_Motion:= Enable_Motion ,
			Enable_Latch:= TRUE,					(*Enabling Runs Valve as detent type (maintained solenoids*)
			Enable_SideA_PreCharge:= FALSE,		(*Enabling Turns Side A PreCharge Active, reset when Side B is energized in Auto*)
			Enable_SideB_PreCharge:= FALSE,		(*Enabling Turns Side B PreCharge Active, reset when Side A is energized in Auto*)
			PreCharge_Time:= T#0.10S,
			Enable_Auto_Commands:= In_Auto,
			Enable_Manual_Commands:= In_Manual AND All_Robots_Clear,
			In_Manual_SideA_Command:= Discrete_In.ManReqs3.28,
			In_Manual_SideB_Command:= Discrete_In.ManReqs3.29,
			SideA_Indicator:= FALSE,
			SideB_Indicator:= FALSE,
			TurnOn_SideA_SOL=> N102.Q.28,
			TurnOn_SideB_SOL=> N102.Q.29,
			TurnOn_SideA_Indicator=> Manual_Indicators3.28,
			TurnOn_SideB_Indicator=> Manual_Indicators3.29
			 );
		Valve47FB.In_Auto_SideA_Command:= FALSE;
		Valve47FB.In_Auto_SideB_Command:= FALSE;


	(*Valve 48, A+B*)
	(*spare*)
		Valve48FB
			(
			Enable_Motion:= Enable_Motion ,
			Enable_Latch:= TRUE,					(*Enabling Runs Valve as detent type (maintained solenoids*)
			Enable_SideA_PreCharge:= FALSE,		(*Enabling Turns Side A PreCharge Active, reset when Side B is energized in Auto*)
			Enable_SideB_PreCharge:= FALSE,		(*Enabling Turns Side B PreCharge Active, reset when Side A is energized in Auto*)
			PreCharge_Time:= T#0.10S,
			Enable_Auto_Commands:= In_Auto,
			Enable_Manual_Commands:= In_Manual AND All_Robots_Clear,
			In_Manual_SideA_Command:= Discrete_In.ManReqs3.30,
			In_Manual_SideB_Command:= Discrete_In.ManReqs3.31,
			SideA_Indicator:= FALSE,
			SideB_Indicator:= FALSE,
			TurnOn_SideA_SOL=> N102.Q.30,
			TurnOn_SideB_SOL=> N102.Q.31,
			TurnOn_SideA_Indicator=> Manual_Indicators3.30,
			TurnOn_SideB_Indicator=> Manual_Indicators3.31
			 );
		Valve48FB.In_Auto_SideA_Command:= FALSE;
		Valve48FB.In_Auto_SideB_Command:= FALSE;


























(*end*)
END_ACTION

ACTION Xfer_To_UI:
(*Transfer General Status of Fixture and I/O Images for Display On HMI*)
	Discrete_Image.Status:= Status;
	Discrete_Image.CLFaults1:= CLFaults1;
	Discrete_Image.CLFaults2:= CLFaults2;
	Discrete_Image.CLFaults3:= CLFaults3;
	Discrete_Image.CLFaults4:= CLFaults4;
	Discrete_Image.CLFaulted:= CLFaulted;
	Discrete_Image.PPFaults:= PPFaults;
	Discrete_Image.PPFaults1:= PPFaults1;
	Discrete_Image.PPFaults2:= PPFaults2;
	Discrete_Image.PPFaulted:= PPFaulted;
	Discrete_Image.Model_Data:= Model_ID;
	Discrete_Image.ToolID:= Fix_ID;
	Discrete_Image.ProdCount:= Prod_Count_Out ;
	Discrete_Image.CycleTime:= Cycle_Time_Out;
	Discrete_Image.PrevCycleTime:= PrevCycle_Time_Out;
	Discrete_Image.LoadTime:= Load_Time_Out;
	Discrete_Image.WeldTime:= Weld_Time_Out;
	Discrete_Image.UnloadTime:= Unload_Time_Out;

	Discrete_Image.InAuto:= In_Auto_Mode;
	Discrete_Image.InManual:= In_Manual_Mode;
	Discrete_Image.ManInds:= Manual_Indicators1;
	Discrete_Image.ManInds2:= Manual_Indicators2;
	Discrete_Image.ManInds3:= Manual_Indicators3;
	Discrete_Image.At_Home:= Tool_At_Home;
	Discrete_Image.Enable_Motion:= Enable_Motion;
	Discrete_Image.All_Sensors_Off:= All_Sensors_Off;
	Discrete_Image.Bypass_ACKS:= Discrete_In.Bypass_REQS;
	Discrete_Image.CustomApplication_ACKS:= Discrete_In.CustomApplication_REQS;
	Discrete_Image.Fixture_Allow_Model_Change:= Fixture_Allow_Model_Change;


	(*See Below for Overiding code as well*)
	Discrete_Image.NodeLayout:=NodeLayout;
	Discrete_Image.NodeState:=NodeState;
	(*
	Overiding code!!!!
	All Nodes after Valve Banks are in Hot connect groups and are for sub fixtures which are interchangable
	Therefore we must decide which node types will be built into the NodeLayout based on model selection
	We must also move the selected Node states as well
	Once everything is moved, then we wll blank out the areas afterward
	*)
	IF Model_ID = 1 OR Model_ID = 2	THEN
		(*Model 504 (1) and Model 524(2) uses Nodes 31/32, whihc are at [34]/[35]*)
		(*Selected Nodes are already at proper array section, blank the rest*)
		Blank_NodeLayout(36);

	ELSIF Model_ID = 3 THEN
		(*Model 543 (3) uses Nodes 42/43, which are at [44]/[45]*)
		Discrete_Image.NodeLayout.NodeName[34]:= NodeLayout.NodeName[44];
		Discrete_Image.NodeLayout.NodeName[35]:= NodeLayout.NodeName[45];
		Discrete_Image.NodeLayout.NodeType[34]:= NodeLayout.NodeType[44];
		Discrete_Image.NodeLayout.NodeType[35]:= NodeLayout.NodeType[45];
		Discrete_Image.NodeState[34]:= NodeLayout.State[44];
		Discrete_Image.NodeState[35]:= NodeLayout.State[45];
		(*Selected Nodes moved to proper array section, blank the rest*)
		Blank_NodeLayout(36);

	ELSIF Model_ID = 4 THEN
		(*Model 526 (4) uses Nodes 40/41, which are at [42]/[43]*)
		Discrete_Image.NodeLayout.NodeName[34]:= NodeLayout.NodeName[42];
		Discrete_Image.NodeLayout.NodeName[35]:= NodeLayout.NodeName[43];
		Discrete_Image.NodeLayout.NodeType[34]:= NodeLayout.NodeType[42];
		Discrete_Image.NodeLayout.NodeType[35]:= NodeLayout.NodeType[43];
		Discrete_Image.NodeState[34]:= NodeLayout.State[42];
		Discrete_Image.NodeState[35]:= NodeLayout.State[43];
		(*Selected Nodes moved to proper array section, blank the rest*)
		Blank_NodeLayout(36);
		
	ELSIF Model_ID = 5 THEN
		(*Model 536 (5) uses Nodes 38/39, which are at [40]/[41]*)
		Discrete_Image.NodeLayout.NodeName[34]:= NodeLayout.NodeName[40];
		Discrete_Image.NodeLayout.NodeName[35]:= NodeLayout.NodeName[41];
		Discrete_Image.NodeLayout.NodeType[34]:= NodeLayout.NodeType[40];
		Discrete_Image.NodeLayout.NodeType[35]:= NodeLayout.NodeType[41];
		Discrete_Image.NodeState[34]:= NodeLayout.State[40];
		Discrete_Image.NodeState[35]:= NodeLayout.State[41];
		(*Selected Nodes moved to proper array section, blank the rest*)
		Blank_NodeLayout(36);

	ELSIF Model_ID = 6 THEN
		(*Model 550 (6) uses Nodes 36/37, which are at [38]/[39]*)
		Discrete_Image.NodeLayout.NodeName[34]:= NodeLayout.NodeName[38];
		Discrete_Image.NodeLayout.NodeName[35]:= NodeLayout.NodeName[39];
		Discrete_Image.NodeLayout.NodeType[34]:= NodeLayout.NodeType[38];
		Discrete_Image.NodeLayout.NodeType[35]:= NodeLayout.NodeType[39];
		Discrete_Image.NodeState[34]:= NodeLayout.State[38];
		Discrete_Image.NodeState[35]:= NodeLayout.State[39];
		(*Selected Nodes moved to proper array section, blank the rest*)
		Blank_NodeLayout(36);

	ELSIF Model_ID = 7 THEN
		(*Model 571 (7) uses Nodes 34/35, which are at [36]/[37]*)
		Discrete_Image.NodeLayout.NodeName[34]:= NodeLayout.NodeName[36];
		Discrete_Image.NodeLayout.NodeName[35]:= NodeLayout.NodeName[37];
		Discrete_Image.NodeLayout.NodeType[34]:= NodeLayout.NodeType[36];
		Discrete_Image.NodeLayout.NodeType[35]:= NodeLayout.NodeType[37];
		Discrete_Image.NodeState[34]:= NodeLayout.State[36];
		Discrete_Image.NodeState[35]:= NodeLayout.State[37];
		(*Selected Nodes moved to proper array section, blank the rest*)
		Blank_NodeLayout(36);
		
	ELSE
		(*No Model means no nodes selected, blank 'em all!*)
		Blank_NodeLayout(34);
	
	END_IF;
		
	
	Discrete_Image.Input_Node_Count:= Discrete_In.Input_Node_Count;
	Discrete_Image.VB_Node_Count:= Discrete_In.VB_Node_Count;
	Discrete_Image.Water_Stand_Count:= Discrete_In.Water_Stand_Count;

	IF  (Discrete_Image.Input_Node_Count < 4)
		THEN Discrete_Image.VB_Screen_Position:= 1;
	ELSIF  (Discrete_Image.Input_Node_Count < 7)
		THEN Discrete_Image.VB_Screen_Position:= 2;
	ELSIF  (Discrete_Image.Input_Node_Count < 10)
		THEN Discrete_Image.VB_Screen_Position:= 3;
	ELSIF  (Discrete_Image.Input_Node_Count < 13)
		THEN Discrete_Image.VB_Screen_Position:= 4;
	ELSIF  (Discrete_Image.Input_Node_Count < 16)
		THEN Discrete_Image.VB_Screen_Position:= 5;
	ELSIF  (Discrete_Image.Input_Node_Count < 19)
		THEN Discrete_Image.VB_Screen_Position:= 6;
	ELSIF  (Discrete_Image.Input_Node_Count < 22)
		THEN Discrete_Image.VB_Screen_Position:= 7;
	ELSIF  (Discrete_Image.Input_Node_Count < 26)
		THEN Discrete_Image.VB_Screen_Position:= 8;
	ELSE
			Discrete_Image.VB_Screen_Position:= 9;
	END_IF;

	Discrete_Image.N00:= N00;
	Discrete_Image.N01:= N01;
	Discrete_Image.N02:= N02;
	Discrete_Image.N03:= N03;
	Discrete_Image.N04:= N04;
	Discrete_Image.N05:= N05;
	Discrete_Image.N06:= N06;
	Discrete_Image.N07:= N07;
	Discrete_Image.N08:= N08;
	Discrete_Image.N09:= N09;
	Discrete_Image.N10:= N10;
	Discrete_Image.N11:= N11;
	Discrete_Image.N12:= N12;
	Discrete_Image.N13:= N13;
	Discrete_Image.N14:= N14;
	Discrete_Image.N15:= N15;
	Discrete_Image.N16:= N16;
	Discrete_Image.N17:= N17;
	Discrete_Image.N18:= N18;
	Discrete_Image.N19:= N19;
	Discrete_Image.N20:= N20;
	Discrete_Image.N21:= N21;
	Discrete_Image.N22:= N22;
	Discrete_Image.N23:= N23;
	Discrete_Image.N24:= N24;
	Discrete_Image.N25:= N25;
	Discrete_Image.N26:= N26;
	Discrete_Image.N27:= N27;
	Discrete_Image.N28:= N28;
	Discrete_Image.N29:= N29;
	Discrete_Image.N30:= N30;
	Discrete_Image.N31:= N31;
	Discrete_Image.N32:= N32;
	Discrete_Image.N33:= N33;
	Discrete_Image.N34:= N34;
	Discrete_Image.N35:= N35;
	Discrete_Image.N36:= N36;
	Discrete_Image.N37:= N37;
	Discrete_Image.N38:= N38;
	Discrete_Image.N39:= N39;
	Discrete_Image.N40:= N40;
	Discrete_Image.N41:= N41;
	Discrete_Image.N42:= N42;
	Discrete_Image.N43:= N43;
	Discrete_Image.N100:= N100;
	Discrete_Image.N100_STAT:= N100_STAT;
	Discrete_Image.N101:= N101;
	Discrete_Image.N101_STAT:= N101_STAT;
	Discrete_Image.N102:= N102;
	Discrete_Image.N102_STAT:= N102_STAT;


	Discrete_Image.ECatSlave_Cable_Breaks:= ECatSlave_Cable_Breaks;

	Discrete_Image.Operator_Performance_Pen:= Production_Report.Shift_Report[0].Prod_Performance;
END_ACTION

END_PROGRAM

// ---- POUs/FBs/FB_TripleCylinder_20150625.TcPOU
(*FB for trpipel sensor, three position, 3 port cylinder":
	Original Author(s): Brent Lekx-Toniolo
------------------------------------------------------------------------------------------
REVISION NOTES:
	Version 20150625
		- Initial Concept, blt
------------------------------------------------------------------------------------------
*)


FUNCTION_BLOCK FB_TripleCylinder_20150625

	VAR_INPUT
		Enable_FB: BOOL;
		Advanced_Sensor: BOOL;
		Retracted_Sensor: BOOL;
		Mid_Sensor: BOOL;
		Advance_Solenoid: BOOL;
		Retract_Solenoid: BOOL;
		Mid_Solenoid: BOOL;
		Adv_Delay: TIME;
		Ret_Delay: TIME;
		Mid_Delay: TIME;
		Fault_Delay: TIME;
		Disable_Fault: BOOL;
	END_VAR

	VAR
		At_Advanced: BOOL;
		At_Retracted: BOOL;
		At_Mid: BOOL;
		Adv_Delay_TMR: TON;
		Ret_Delay_TMR: TON;
		Mid_Delay_TMR: TON;
		Sensor_FLT_TMR: TON;
		Advancing_FLT_TMR: TON;
		Retracting_FLT_TMR: TON;
		Middling_FLT_TMR: TON;
	END_VAR

	VAR_OUTPUT
		FB_OK: BOOL;
		In_Advanced_Position: BOOL;
		In_Retracted_Position: BOOL;
		In_Mid_Position: BOOL;
		Faulted: BOOL;
		Sensor_Fault: BOOL;
		Advancing_Fault: BOOL;
		Retracting_Fault: BOOL;
		Middling_Fault: BOOL;
	END_VAR

	(*Set FB_OK to True*)
	FB_OK:= TRUE;
(*$$$$$$$$$$$$$$$$$$$$$$$$$$$$$$$$$$ Internal Code $$$$$$$$$$$$$$$$$$$$$$$$$$$$$$$$$$$$$$$$$$$$$$$*)
	(*Develop Advanced Position*)
	At_Advanced:= Advanced_Sensor AND NOT Mid_Sensor AND NOT Retracted_Sensor;

	(*Develop Retracted Position*)
	At_Retracted:= Retracted_Sensor AND NOT Mid_Sensor AND NOT Advanced_Sensor;

	(*Develop Mid Position*)
	At_Mid:= Mid_Sensor AND NOT Advanced_Sensor AND NOT Retracted_Sensor;

	(*Delay Advanced Position Output*)
	Adv_Delay_TMR.PT:= Adv_Delay;
	Adv_Delay_TMR.IN:= At_Advanced;
	Adv_Delay_TMR();
	In_Advanced_Position:= Adv_Delay_TMR.Q;

	(*Delay Retracted Position Output*)
	Ret_Delay_TMR.PT:= Ret_Delay;
	Ret_Delay_TMR.IN:= At_Retracted;
	Ret_Delay_TMR();
	In_Retracted_Position:= Ret_Delay_TMR.Q;

	(*Delay Mid Position Output*)
	Mid_Delay_TMR.PT:= Mid_Delay;
	Mid_Delay_TMR.IN:= At_Mid;
	Mid_Delay_TMR();
	In_Mid_Position:= Mid_Delay_TMR.Q;

(*$$$$$$$$$$$$$$$$$$$$$$$$$$$$$$$$$$$$$$$$ Fault Code $$$$$$$$$$$$$$$$$$$$$$$$$$$$$$$$$$$$$$$$$$$$$$$$*)
	(*Sensor Fault*)
	Sensor_FLT_TMR.PT:= Fault_Delay;
	Sensor_FLT_TMR.IN:= (NOT At_Advanced AND NOT At_Mid AND NOT At_Retracted)
						OR (At_Advanced AND At_Retracted)
						OR (At_Advanced AND At_Mid)
						OR (At_Mid AND At_Retracted);
	Sensor_FLT_TMR();
	Sensor_Fault:= Sensor_FLT_TMR.Q;

	(*Advancing Fault*)
	Advancing_FLT_TMR.PT:= Fault_Delay;
	Advancing_FLT_TMR.IN:= Advance_Solenoid AND NOT At_Advanced AND NOT Sensor_Fault;
	Advancing_FLT_TMR();
	Advancing_Fault:= Advancing_FLT_TMR.Q;

	(*Retracting Fault*)
	Retracting_FLT_TMR.PT:= Fault_Delay;
	Retracting_FLT_TMR.IN:= Retract_Solenoid AND NOT Mid_Solenoid AND NOT At_Retracted AND NOT Sensor_Fault;
	Retracting_FLT_TMR();
	Retracting_Fault:= Retracting_FLT_TMR.Q;

	(*Middling Fault*)
	Middling_FLT_TMR.PT:= Fault_Delay;
	Middling_FLT_TMR.IN:= Mid_Solenoid AND NOT Advance_Solenoid AND NOT At_Mid AND NOT Sensor_Fault;
	Middling_FLT_TMR();
	Middling_Fault:= Middling_FLT_TMR.Q;

	(*Develop Fault Output*)
	Faulted:=NOT Disable_Fault AND  (Sensor_Fault OR Advancing_Fault OR Middling_Fault OR Retracting_Fault);

END_FUNCTION_BLOCK

// ---- POUs/FBs/FB_GTAC_QAcheck_20150529.TcPOU
(*FB for use as framework for Nut Checnk type functions:
	Original Author(s): Rob Remillard of Sodecia GTAC; 
------------------------------------------------------------------------------------------
REVISION NOTES:
	Version: 20130620
	- Original Concept, r.remillard
	Version: 20150130
	- Change all naming from "Nut...." to QA....." for more generic uses, b.toniolo/r.remillard
	Version 20150210
	- Changed Not Ok Reset routine, r.remillard and b.lekx-toniolo
	Version 20150529
	- added QAcheck_release, jvd
	-changed QAcheck_Reset2 to be QAcheck_Retry, jvd
	- QA check FB now has a retry option or a release option, in the instance put the reset condition to either input, jvd
------------------------------------------------------------------------------------------
*)

FUNCTION_BLOCK FB_GTAC_QAcheck_20150529

VAR_INPUT

	Start_QAcheck:						BOOL;
	QAcheck_Reset:						BOOL;
	QAcheck_Retry:						BOOL;
	QAcheck_Release:					BOOL;

	QAcheck_Adv_In:						BOOL;
	QAcheck_Ret_In:						BOOL;

	User_Dry_Cycle:						BOOL;

	QAcheck_OK_Delay:					TIME;
	QAcheck_Fault_Delay:					TIME;

END_VAR

VAR_OUTPUT

	QAcheck_OK:						BOOL;
	QAcheck_Failed:						BOOL;
	Fire_QAchecks:						BOOL;

END_VAR


VAR
	QAcheck_OK_Time:					TON;
	QAcheck_Fault_Time:					TON;

END_VAR

(*Move Delay times into timers*)
	QAcheck_OK_Time.PT:= QAcheck_OK_Delay;
	QAcheck_OK_Time();
	QAcheck_Fault_Time.PT:= QAcheck_Fault_Delay;
	QAcheck_Fault_Time();


(*Tigger QA Check*)
IF Start_QAcheck AND NOT QAcheck_OK AND NOT QAcheck_Reset
	THEN
		Fire_QAchecks:= TRUE;
ELSE
		Fire_QAchecks:= FALSE;

END_IF;


(*QA Check OK Routine*)
IF ((Start_QAcheck AND QAcheck_Adv_In) OR QAcheck_OK OR (User_Dry_Cycle AND NOT QAcheck_Ret_In))
     	AND NOT QAcheck_Reset  AND NOT QAcheck_Failed
	THEN
		QAcheck_OK_Time.IN:= TRUE;
		IF QAcheck_OK_Time.Q
			THEN
				QAcheck_OK:= TRUE;
		END_IF;

ELSE
		QAcheck_OK:= FALSE;
		QAcheck_OK_Time.IN:= FALSE;
END_IF;

IF QAcheck_Release  AND QAcheck_Failed
	THEN
	QAcheck_OK := TRUE;
	QAcheck_Failed := FALSE;
END_IF;


(*QA Check NOT OK Routine*)
IF (Start_QAcheck AND NOT QAcheck_OK OR QAcheck_Failed)
      AND NOT QAcheck_Retry  AND NOT User_Dry_Cycle
	THEN
		QAcheck_Fault_Time.IN:= TRUE;
		IF QAcheck_Fault_Time.Q
			THEN
				QAcheck_Failed:= TRUE;
		END_IF;
ELSE
		QAcheck_Failed:= FALSE;
		QAcheck_Fault_Time.IN:= FALSE;
END_IF;

END_FUNCTION_BLOCK

// ---- POUs/FBs/FB_GTAC_Load_Seq_20230302.TcPOU
(*FB for use Fixture Load sequences:
	Original Author(s): Justin Vandongen of Sodecia GTAC; 
------------------------------------------------------------------------------------------
REVISION NOTES:
	Version 20180305
		- Initial Concept, j.vandongen
	Version 20200130
		- updated fault code, j.vandongen
	Version
		- latched on load sequence bits unless timer is elasped, j.vandongen
	Version 20230302
		- Changed declaration of Load-Sequence variable to persistent type as per request detailed in GH Issue #8 in 5.06, b.lekx-toniolo
------------------------------------------------------------------------------------------
*)

FUNCTION_BLOCK FB_GTAC_Load_Seq_20230302
	VAR_INPUT
		Enable_Motion: BOOL;
		Seq_Steps: UDINT;

		Stage1_Check: BOOL;
		Stage2_Check: BOOL;
		Stage3_Check: BOOL;

		Reset: BOOL;
		Disable_Faults: BOOL;
	END_VAR
	
	
	VAR_OUTPUT
		FB_OK: BOOL;
		Faulted: BOOL;
		Load_SequenceOK: BOOL;

		Stage1_TMR: TON;
		Stage2_TMR: TON;
		Stage3_TMR: TON;

	END_VAR
	

	VAR PERSISTENT
		
	(*Standard Internals*)
		Load_Sequence: UDINT;

	END_VAR

	(*Set FB_OK to True*)
	FB_OK:= TRUE;


(*$$$$$$$$$$$$$$$$$$$$$$$$$$$$$$$$$$$$$$$$$$$$$ Internal Code $$$$$$$$$$$$$$$$$$$$$$$$$$$$$$$$$$$$$$$$$$$$$$$$$$$$$$$$$*)
	(*First Stage*)
	IF Stage1_Check AND NOT Stage2_Check AND NOT Stage3_Check
		THEN
			Load_Sequence.0:= TRUE;
	ELSIF NOT Stage1_Check AND NOT Disable_Faults AND Stage1_TMR.Q
		THEN
			Load_Sequence.0:= FALSE;
	END_IF;

	(*If Stage 1 shuts off, wait a time and then allow fault. stage check debounce*)
	Stage1_TMR(
			IN:= Load_Sequence.0 AND NOT Stage1_Check ,
			PT:= T#750ms,
			Q=> ,
			ET=> );



	(*Second Stage*)
	IF Load_Sequence.0 AND Stage2_Check AND NOT Stage3_Check
		THEN
			Load_Sequence.1:= TRUE;
	ELSIF (NOT Stage1_Check OR NOT Stage2_Check) AND NOT Disable_Faults  AND Stage2_TMR.Q
		THEN
			Load_Sequence.1:= FALSE;
	END_IF;

	(*If Stage 2 shuts off, wait a time and then allow fault. stage check debounce*)
	Stage2_TMR(
			IN:= Load_Sequence.1 AND NOT Stage2_Check ,
			PT:= T#750ms,
			Q=> ,
			ET=> );



	(*Third Stage*)
	IF Load_Sequence.1 AND Stage3_Check
		THEN
			Load_Sequence.2:= TRUE;
	ELSIF (NOT Stage1_Check OR NOT Stage2_Check OR NOT Stage3_Check) AND NOT Disable_Faults AND Stage3_TMR.Q
		THEN
			Load_Sequence.2:= FALSE;
	END_IF;

	(*If Stage 3 shuts off, wait a time and then allow fault. stage check debounce*)
	Stage3_TMR(
			IN:= Load_Sequence.2 AND NOT Stage3_Check ,
			PT:= T#750ms,
			Q=> ,
			ET=> );



(*$$$$$$$$$$$$$$$$Gather all Load Sequences$$$$$$$$$$$$$$$$*)
	(*Load Sequence OK*)
	IF (Stage1_Check AND Load_Sequence.0)
		AND (Stage2_Check AND Load_Sequence.1)
		AND ((Stage3_Check AND Load_Sequence.2)  OR (Seq_Steps=2))
		AND NOT Faulted
		THEN
			Load_SequenceOK:= TRUE;
	END_IF;



(*$$$$$$$$$$$$$$$$Gather all Load Sequence Faults$$$$$$$$$$$$$$$$*)
	(*Fault Logic*)
	IF ((NOT Stage1_Check AND (Stage2_Check OR Stage3_Check))
		OR (Stage1_Check AND (Stage2_Check OR Stage3_Check) AND NOT Load_Sequence.0)
		OR (Stage1_Check AND NOT Stage2_Check AND Stage3_Check))
		AND NOT Disable_Faults
		THEN
			Load_SequenceOK:= FALSE;
			Faulted:= TRUE;
	END_IF;



(*$$$$$$$$$$$$$$$$Reset all Load Sequences$$$$$$$$$$$$$$$$*)
	(*Reset Load Sequence*)
	IF Reset
		THEN
			Load_Sequence:= 0;
			Load_SequenceOK:= FALSE;
			Faulted:= FALSE;
	END_IF;






















(*end*)

END_FUNCTION_BLOCK

// ---- POUs/FBs/FB_Production_Report_20221007.TcPOU
(*FB FOR use to generate OEE based Data production reports for a 1-3 shift manufacturing facility with ability to configure shift structure.


	Original Author(S): Rob Remillard and Brent Lekx-Toniolo of Sodecia GTAC
------------------------------------------------------------------------------------------
	REVISION NOTES:
	DATE: 2008
	- original concept, r.remillad and b.lekx-toniolo
	Version 20141030:
	- Changed name to include date stamped version control
	- Added Element [0] to Shift Report Array and code to dump curent data to this element, b.lekx-toniolo
	Version 20150819:
	- Re-typed Variables "Production_Count" and "Running_Target _Count" from INT to UNIT to avoid compiler warnings, b.lekx-toniolo
	Version 20160229
		- Updated shift report udt instance, b.lekx-toniolo
	Version 20160513
		- Changed Reporting structure so that only Report[0] was curent, all others were kept until shift end, b.lekx-toniolo
	Version 20160519
		- Added Configurability to shift structures, b.lekx-toniolo		
	Version 20191125
		- Changes / Additions during 2019 production reporting code upgrades (for config via UI), b.lekx-toniolo		
	Version 20221007
		- Uopdates to report udt to add in Target_Cycle_Time to report capturing, b.lekx-toniolo	
	Version 20252801
		- Added Shift Letter to code - starts Line 114, r.jones

------------------------------------------------------------------------------------------
*)



FUNCTION_BLOCK FB_Production_Report_20221007
VAR_INPUT
	Enable_FB: BOOL;
	StartEnd_Mode: UINT;
	Manual_Start: BOOL;
	Manual_End: BOOL;
	Prod_Inc: BOOL;
	Scrap_Inc: BOOL;
	Scrap_Dec: BOOL;
	Reference_TimeDate: TimeStruct;
	Reference_Target_Time: TIME;
	Enable_InShift_Change: BOOL;

	Config_Day_TOD: udt_Generic_ShiftConfigTOD_20160527;
	Config_Aft_TOD: udt_Generic_ShiftConfigTOD_20160527;
	Config_Mid_TOD: udt_Generic_ShiftConfigTOD_20160527;
	Config_Shift_Enables: UINT;		(*Enable Flags for shifts in a 24 hour period*)
	Config_Break_Count: UINT;			(*Amount of breaks per shift*)

	Static_Target: UINT;
	Machine_Serial: STRING;
	Machine_Common_Name: STRING;
	Operator_ID: UINT;
	Model_Data:UINT;
	Fix_ID: UINT;
	Machine_StoppedBy_Fault: BOOL;
	Test_Start: BOOL;
	Test_End: BOOL;

END_VAR
VAR
	Report_In_Auto: BOOL;
	Report_In_Override: BOOL;
	Reference_Time_TOD: TOD;
	Config_Day: udt_Generic_ShiftConfig_20160519;
	Config_Aft: udt_Generic_ShiftConfig_20160519;
	Config_Mid: udt_Generic_ShiftConfig_20160519;
		Day_Shift_ConfigOK: BOOL;
		Mid_Shift_ConfigOK: BOOL;
		Aft_Shift_ConfigOK: BOOL;

		Day_Shift_Enabled: BOOL;
		Aft_Shift_Enabled: BOOL;
		Mid_Shift_Enabled: BOOL;
		Break1_Enabled: BOOL;
		Break2_Enabled: BOOL;
		Break3_Enabled: BOOL;


	Shift_Report: ARRAY [0..3] OF udt_Generic_Production_20221007;

	In_Day_Shift: BOOL;
	In_Aft_Shift: BOOL;
	In_Mid_Shift: BOOL;
	In_Shift_Code: UINT;
	In_Hour_Code: UINT;
	In_Break: BOOL;
	In_Shift_Change: BOOL;
	Machine_Running: BOOL;

	Running_Difference: DINT;

	Running_TotalTime: TIME;
	Running_TotalBy_Expected: REAL;
	Running_UpTime: TIME;
	Running_AvailabilityEFF: REAL;
	Running_PerformanceEFF: REAL;
	Running_QualityEFF: REAL;
	Running_OEE: REAL;

	Start_Shift_Trigger: R_TRIG;
	Hourly_Trigger: R_TRIG;
	End_Shift_Trigger: R_TRIG;
	Target_Trigger: R_TRIG;
	FaultCount_Inc_Trigger: R_TRIG;
	Not_Faulted_Trigger: R_TRIG;
	Scrap_Inc_Trigger:R_TRIG;
	Scrap_Dec_Trigger:R_TRIG;

	Target_TMR: TON;
	Faulted_TMR: TON;
	Status: STRING;
	Gross_Shift_Duration: REAL;
	Net_Shift_Duration: REAL;

END_VAR

VAR PERSISTENT
	Production_Count: UINT;
	Running_Target_Count: UINT;
	Running_Target_CountPrevHourTotal: UINT;
	Running_Scrap_Count: UINT;
	Total_Faulted_Time: TIME;
	Previous_Faulted_Time: TIME;
	Total_Fault_Count: UDINT;
	PartsLost_From_Faults: REAL;

END_VAR


VAR_OUTPUT
	FB_Ok: BOOL;
	Shift_Letter : STRING[1] ;
END_VAR

(*---------------------------------------------------Type Converstions to allow both type of time formats to be avalable -----------------------------------*)

(*Convert Shift Report Structrues from TOD to OTStruct*)

	ShiftConfigs_TOD_To_OTSTRUCT();

(*Convert Reference Time to TOD Type*)
 	Reference_Time_TOD:= FUN_GTAC_TIMESTRUCTtoTOD(Reference_TimeDate);

(*------------------------------------------------------ Check for some basics on Config Information --------------------------------------------------------------------*)

	(*Check some general validity to shift configuratons (MAY NOT CATCH ALL CONFIG MISTAKES)*)
	(*Set FB_OK to True*)
		Day_Shift_ConfigOK:=  ((Config_Day_TOD.Shift_StartTime < Config_Day_TOD.Shift_EndTime
			AND ((Config_Day_TOD.Break1_StartTime < Config_Day_TOD.Break1_EndTime) OR NOT Break1_Enabled)
			AND ((Config_Day_TOD.Break2_StartTime < Config_Day_TOD.Break2_EndTime) OR NOT Break2_Enabled)
			AND ((Config_Day_TOD.Break3_StartTime < Config_Day_TOD.Break3_EndTime) OR NOT Break3_Enabled))
			OR NOT Day_Shift_Enabled);

		Aft_Shift_ConfigOK:= ((Config_Aft_TOD.Shift_StartTime <Config_Aft_TOD.Shift_EndTime
			AND ((Config_Aft_TOD.Break1_StartTime < Config_Aft_TOD.Break1_EndTime) OR NOT Break1_Enabled)
			AND ((Config_Aft_TOD.Break2_StartTime < Config_Aft_TOD.Break2_EndTime) OR NOT Break2_Enabled)
			AND ((Config_Aft_TOD.Break3_StartTime < Config_Aft_TOD.Break3_EndTime) OR NOT Break3_Enabled))
			OR NOT Aft_Shift_Enabled);

		Mid_Shift_ConfigOK:= ((Config_Mid_TOD.Shift_StartTime > Config_Mid_TOD.Shift_EndTime (*Midnight Shift must fall over the midnight change*)
			AND(
				(((((Config_Mid_TOD.Break1_StartTime > TOD#12:00:00 AND Config_Mid_TOD.Break1_EndTime >TOD#12:00:00)
					OR
				(Config_Mid_TOD.Break1_StartTime < TOD#12:00:00 AND Config_Mid_TOD.Break1_EndTime <TOD#12:00:00)) AND
					Config_Mid_TOD.Break1_StartTime < Config_Mid_TOD.Break1_EndTime)
				OR ((Config_Mid_TOD.Break1_StartTime > TOD#12:00:00 AND Config_Mid_TOD.Break1_EndTime <TOD#12:00:00) AND Config_Mid_TOD.Break1_StartTime > Config_Mid_TOD.Break1_EndTime))
				OR NOT Break1_Enabled)

			AND (((((Config_Mid_TOD.Break2_StartTime > TOD#12:00:00 AND Config_Mid_TOD.Break2_EndTime >TOD#12:00:00)
					OR
				(Config_Mid_TOD.Break2_StartTime < TOD#12:00:00 AND Config_Mid_TOD.Break2_EndTime <TOD#12:00:00)) AND
					Config_Mid_TOD.Break2_StartTime < Config_Mid_TOD.Break2_EndTime)
				OR ((Config_Mid_TOD.Break2_StartTime > TOD#12:00:00 AND Config_Mid_TOD.Break2_EndTime <TOD#12:00:00) AND Config_Mid_TOD.Break2_StartTime > Config_Mid_TOD.Break2_EndTime))
				OR NOT Break2_Enabled)
			AND (((((Config_Mid_TOD.Break3_StartTime > TOD#12:00:00 AND Config_Mid_TOD.Break3_EndTime >TOD#12:00:00)
					OR
				(Config_Mid_TOD.Break3_StartTime < TOD#12:00:00 AND Config_Mid_TOD.Break3_EndTime <TOD#12:00:00)) AND
					Config_Mid_TOD.Break3_StartTime < Config_Mid_TOD.Break3_EndTime)
				OR ((Config_Mid_TOD.Break3_StartTime > TOD#12:00:00 AND Config_Mid_TOD.Break3_EndTime <TOD#12:00:00) AND Config_Mid_TOD.Break3_StartTime > Config_Mid_TOD.Break3_EndTime))
				OR NOT Break3_Enabled)
				))

			OR NOT Mid_Shift_Enabled);



(*Develop FB_OK from above*)

	FB_OK:= Day_Shift_ConfigOK AND
			Aft_Shift_ConfigOK AND
			Mid_Shift_ConfigOK;

(*----------------------------------------------------- Decode Shift and Break Enables --------------------------------------------------------------------------------------------------*)

	Day_Shift_Enabled:= Config_Shift_Enables.1 AND FB_OK;
	Aft_Shift_Enabled:= Config_Shift_Enables.2 AND FB_OK;
	Mid_Shift_Enabled:= Config_Shift_Enables.3 AND FB_OK;


	Break1_Enabled:= (Config_Break_Count>=1) AND (Config_Shift_Enables>0) AND FB_OK;
	Break2_Enabled:= (Config_Break_Count>=2) AND (Config_Shift_Enables>0) AND FB_OK;
	Break3_Enabled:= (Config_Break_Count>=3) AND (Config_Shift_Enables>0) AND FB_OK;


(*------------------------------------------------------------------------------------------ Production Report FB ---------------------------------------------------------------------------*)

(*Determine Shift Report Mode*)

	(*Report In Auto, So Start Stop at Shift Change*)
	IF StartEnd_Mode=0
		THEN
			Report_In_Auto:= TRUE;
			Report_In_Override:= FALSE;
	END_IF;

	(*Report In Override, So Start and Stop Given By Operator*)
	IF StartEnd_Mode=1
		THEN
			Report_In_Auto:= FALSE;
			Report_In_Override:= TRUE;
	END_IF;

(*------------------------------------------------------------- Calculate Shift Duration Times ----------------------------------------------------------------*)

	IF In_Day_Shift
		THEN
		Gross_Shift_Duration:= FUN_GTAC_ReturnGrossShiftDuration(Config_Day_TOD);
		Net_Shift_Duration:= FUN_GTAC_ReturnNetShiftDuration(Config_Day_TOD, Config_Break_Count);
	ELSIF In_Aft_Shift
		THEN
		Gross_Shift_Duration:= FUN_GTAC_ReturnGrossShiftDuration(Config_Aft_TOD);
		Net_Shift_Duration:= FUN_GTAC_ReturnNetShiftDuration(Config_Aft_TOD, Config_Break_Count);
	ELSIF In_Mid_Shift
		THEN
		Gross_Shift_Duration:= FUN_GTAC_ReturnGrossShiftDuration(Config_Mid_TOD);
		Net_Shift_Duration:= FUN_GTAC_ReturnNetShiftDuration(Config_Mid_TOD, Config_Break_Count);
	END_IF;

(* Subtract 10 minutes for In Shift Change (5 minutes at start and end of shift) if enabled*)
	IF Enable_InShift_Change AND (In_Day_Shift OR In_Aft_Shift OR In_Mid_Shift)
		THEN
			Net_Shift_Duration:= Net_Shift_Duration - 0.1666666; (*Subtract a total of 10 minutes from shift (10/60)*)
	END_IF;

(*------------------------------------------------------------------------- Shift Report Auto Mode Code -------------------------------------------------------*)

	(*In Day Shift*)
	IF Day_Shift_Enabled AND
		Reference_Time_TOD >= Config_Day_TOD.Shift_StartTime AND
		Reference_Time_TOD < Config_Day_TOD.Shift_EndTime
		THEN
			In_Day_Shift:= TRUE;
			In_Aft_Shift:= FALSE;
			In_Mid_Shift:= FALSE;
			In_Shift_Code:=1;
			Shift_Letter := 'A';
	(*In Afternoon Shift*)
	ELSIF Aft_Shift_Enabled AND
			Reference_Time_TOD >= Config_Aft_TOD.Shift_StartTime AND
			Reference_Time_TOD < Config_Aft_TOD.Shift_EndTime
		THEN
			In_Day_Shift:= FALSE;
			In_Aft_Shift:= TRUE;
			In_Mid_Shift:= FALSE;
			In_Shift_Code:=2;
		    Shift_Letter := 'B';
	(*In Midnight Shift*)
	ELSIF Mid_Shift_Enabled AND
			((Reference_Time_TOD <=TOD#23:59:59) AND Reference_Time_TOD >= Config_Mid_TOD.Shift_StartTime)
		 	OR ((Reference_Time_TOD >= TOD#00:00:00) AND Reference_Time_TOD < Config_Mid_TOD.Shift_EndTime)
		THEN
			In_Day_Shift:= FALSE;
			In_Aft_Shift:= FALSE;
			In_Mid_Shift:= TRUE;
			In_Shift_Code:=3;
			Shift_Letter := 'C';
	ELSE
			In_Day_Shift:= FALSE;
			In_Aft_Shift:= FALSE;
			In_Mid_Shift:= FALSE;
			In_Shift_Code:=0;
			Shift_Letter := '';
	END_IF;
(*Perform Limit Check*)
	IF In_Shift_Code<0
		THEN
			In_Shift_Code:=0;
	ELSIF In_Shift_Code>3
		THEN
			In_Shift_Code:=3;
	END_IF;


(*-------------------- Generate Hour Code --------------------*)
(*The hour code is which hour are we into compared to shift start
Examples:
	1. Shift starts at 7:00am, current time is 8:29am. Therefore we are in "Hour 2" (as Hour 1 is 7:00am to 7:59, Hour 2 is 8:00am to 8:59)
	2. Shift starts at 7:30am, current time is 8:29am. Therefore we are in "Hour 1" (as Hour 1 is 7:30am to 8:29, Hour 2 is 8:30am to 9:29)
*)
	IF In_Day_Shift AND Reference_TimeDate.wHour>0
		THEN
			In_Hour_Code:= UDINT_TO_UINT(((TOD_TO_UDINT(Reference_Time_TOD)/60000) - (TOD_TO_UDINT(Config_Day_TOD.Shift_StartTime)/60000))/60+1);
	ELSIF In_Aft_Shift
		THEN
		IF (Reference_TimeDate.wHour >= Config_Aft.Shift_StartTime.wHour)
			THEN
			In_Hour_Code:= UDINT_TO_UINT(((TOD_TO_UDINT(Reference_Time_TOD)/60000) - (TOD_TO_UDINT(Config_Aft_TOD.Shift_StartTime)/60000))/60+1);
		ELSIF (Reference_TimeDate.wHour < Config_Aft.Shift_StartTime.wHour)
			THEN
			In_Hour_Code:= UDINT_TO_UINT((((86400000 - TOD_TO_UDINT(Config_Aft_TOD.Shift_StartTime))/60000) + (TOD_TO_UDINT(Reference_Time_TOD)/60000)) /60+1);
		END_IF;
	ELSIF In_Mid_Shift
		THEN
		IF (Reference_TimeDate.wHour >= Config_Mid.Shift_StartTime.wHour)
			THEN
			In_Hour_Code:= UDINT_TO_UINT(((TOD_TO_UDINT(Reference_Time_TOD)/60000) - (TOD_TO_UDINT(Config_Mid_TOD.Shift_StartTime)/60000))/60+1);
		ELSIF (Reference_TimeDate.wHour < Config_Mid.Shift_StartTime.wHour)
			THEN
			In_Hour_Code:= UDINT_TO_UINT((((86400000 - TOD_TO_UDINT(Config_Mid_TOD.Shift_StartTime))/60000) + (TOD_TO_UDINT(Reference_Time_TOD)/60000)) /60+1);
		END_IF;
	END_IF;
(*Perform Limit Check*)
	IF In_Hour_Code<1
		THEN
			In_Hour_Code:=1;
	ELSIF In_Hour_Code>12
		THEN
			In_Hour_Code:=12;
	END_IF;

(*------------------------- In Break Time------------------------*)

	IF In_Day_Shift AND
				((Reference_Time_TOD >= Config_Day_TOD.Break1_StartTime AND  Reference_Time_TOD < Config_Day_TOD.Break1_EndTime)
				OR (Reference_Time_TOD >= Config_Day_TOD.Break2_StartTime AND  Reference_Time_TOD < Config_Day_TOD.Break2_EndTime)
				OR (Reference_Time_TOD >= Config_Day_TOD.Break3_StartTime AND  Reference_Time_TOD < Config_Day_TOD.Break3_EndTime))
		THEN
		In_Break:= TRUE;
	ELSIF In_Aft_Shift AND
				 ((Reference_Time_TOD >= Config_Aft_TOD.Break1_StartTime AND  Reference_Time_TOD < Config_Aft_TOD.Break1_EndTime)
				OR (Reference_Time_TOD >= Config_Aft_TOD.Break2_StartTime AND  Reference_Time_TOD < Config_Aft_TOD.Break2_EndTime)
				OR (Reference_Time_TOD >= Config_Aft_TOD.Break3_StartTime AND  Reference_Time_TOD < Config_Aft_TOD.Break3_EndTime))
		THEN
		In_Break:= TRUE;
	ELSIF In_Mid_Shift AND
				((Reference_Time_TOD >= Config_Mid_TOD.Break1_StartTime AND  Reference_Time_TOD < Config_Mid_TOD.Break1_EndTime)
				OR (Reference_Time_TOD >= Config_Mid_TOD.Break2_StartTime AND  Reference_Time_TOD < Config_Mid_TOD.Break2_EndTime)
				OR (Reference_Time_TOD >= Config_Mid_TOD.Break3_StartTime AND  Reference_Time_TOD < Config_Mid_TOD.Break3_EndTime))
		THEN
		In_Break:= TRUE;
	ELSE
		In_Break:= FALSE;
	END_IF;

(*---------------------- In Shift Change -----------------------*)
(*If enabled by config, the expected count will cease to take place for a 5 minute period at start and end of shift*)
(*10 minutes is also removed from the machine full running time*)

	IF Enable_InShift_Change AND In_Day_Shift AND
					((Reference_TimeDate.wHour=Config_Day.Shift_StartTime.wHour AND Reference_TimeDate.wMinute>=Config_Day.Shift_StartTime.wMinute AND Reference_TimeDate.wMinute<=Config_Day.Shift_StartTime.wMinute+5)
					OR (Reference_TimeDate.wHour >= Config_Day.Shift_EndTime.wHour-1 AND Reference_Time_TOD > UDINT_TO_TOD(TOD_TO_UDINT(Config_Day_TOD.Shift_EndTime) - 300000)))
		THEN
		In_Shift_Change:= TRUE;
	ELSIF Enable_InShift_Change AND In_Aft_Shift AND
					((Reference_TimeDate.wHour=Config_Aft.Shift_StartTime.wHour AND Reference_TimeDate.wMinute>=Config_Aft.Shift_StartTime.wMinute AND Reference_TimeDate.wMinute<=Config_Aft.Shift_StartTime.wMinute+5)
					OR (Reference_TimeDate.wHour >= Config_Aft.Shift_EndTime.wHour-1 AND Reference_Time_TOD > UDINT_TO_TOD(TOD_TO_UDINT(Config_Aft_TOD.Shift_EndTime) - 300000)))
		THEN
		In_Shift_Change:= TRUE;
	ELSIF Enable_InShift_Change AND In_Mid_Shift AND
					((Reference_TimeDate.wHour=Config_Mid.Shift_StartTime.wHour AND Reference_TimeDate.wMinute>=Config_Mid.Shift_StartTime.wMinute AND Reference_TimeDate.wMinute<=Config_Mid.Shift_StartTime.wMinute+5)
					OR  (((Reference_Time_TOD >= TOD#00:00:00) AND Reference_Time_TOD < Config_Mid_TOD.Shift_EndTime) AND
						(Reference_TimeDate.wHour >= Config_Mid.Shift_EndTime.wHour-1 AND Reference_Time_TOD > UDINT_TO_TOD(TOD_TO_UDINT(Config_Mid_TOD.Shift_EndTime) - 300000))))
		THEN
		In_Shift_Change:= TRUE;
	ELSE
		In_Shift_Change:= FALSE;
	END_IF;

(*------------ Generate Start of Shift, Hourly and End Of Shift Triggers (1 Scan Pulses) ------------*)

	(*Start of Shift Trigger*)
	Start_Shift_Trigger.CLK:= In_Day_Shift AND ((Reference_TimeDate.wHour = Config_Day.Shift_StartTime.wHour AND Reference_TimeDate.wMinute = Config_Day.Shift_StartTime.wMinute) OR Test_Start)
							OR (In_Aft_Shift AND ((Reference_TimeDate.wHour = Config_Aft.Shift_StartTime.wHour AND Reference_TimeDate.wMinute = Config_Aft.Shift_StartTime.wMinute) OR Test_Start))
							OR (In_Mid_Shift AND ((Reference_TimeDate.wHour = Config_Mid.Shift_StartTime.wHour AND Reference_TimeDate.wMinute = Config_Mid.Shift_StartTime.wMinute) OR Test_Start));
	Start_Shift_Trigger();

	(*Hourly Trigger*)
	Hourly_Trigger.CLK:= Reference_TimeDate.wMinute = 0 AND Reference_TimeDate.wSecond = 0;
	Hourly_Trigger();

	(*End of Shift Trigger*)
	End_Shift_Trigger.CLK:= (In_Day_Shift AND Reference_Time_TOD > UDINT_TO_TOD(TOD_TO_UDINT(Config_Day_TOD.Shift_EndTime)-1000))
							OR (In_Aft_Shift AND Reference_Time_TOD > UDINT_TO_TOD(TOD_TO_UDINT(Config_Aft_TOD.Shift_EndTime)-1000))
							OR (In_Mid_Shift AND (Reference_Time_TOD <Config_Mid_TOD.Shift_EndTime) AND Reference_Time_TOD > UDINT_TO_TOD(TOD_TO_UDINT(Config_Mid_TOD.Shift_EndTime)-1000));

	End_Shift_Trigger();


(*----------------------------------------------------- Generate Target Cycle Time ----------------------------------------------------------------------------------------*)

	Target_TMR.PT:= Reference_Target_Time;
	Target_TMR.IN:= (NOT Target_Trigger.Q AND (In_Day_Shift OR In_Aft_Shift OR In_Mid_Shift));
	Target_TMR();

(*------------------ Generate Running Target Time Trigger ---------------*)

	Target_Trigger.CLK:= Target_TMR.Q;
	Target_Trigger();

(*----------------- Generate Running Target ---------------------------*)

	IF Target_Trigger.Q AND NOT In_Break AND NOT In_Shift_Change
		THEN
			Running_Target_Count:= Running_Target_Count+1;
	END_IF;

(*Track Running Target Count for Use in Calcing Hourly TargetCount*)
	IF NOT Hourly_Trigger.Q
		THEN
		IF In_Hour_Code=1
			THEN
				Running_Target_CountPrevHourTotal:= 0;
		ELSIF In_Hour_Code=2
			THEN
				Running_Target_CountPrevHourTotal:= Shift_Report[0].Expected_Count[1];
		ELSIF In_Hour_Code=3
			THEN
				Running_Target_CountPrevHourTotal:= Shift_Report[0].Expected_Count[1]+
													Shift_Report[0].Expected_Count[2];
		ELSIF In_Hour_Code=4
			THEN
				Running_Target_CountPrevHourTotal:= Shift_Report[0].Expected_Count[1]+
													Shift_Report[0].Expected_Count[2]+
													Shift_Report[0].Expected_Count[3];
		ELSIF In_Hour_Code=5
			THEN
				Running_Target_CountPrevHourTotal:= Shift_Report[0].Expected_Count[1]+
													Shift_Report[0].Expected_Count[2]+
													Shift_Report[0].Expected_Count[3]+
													Shift_Report[0].Expected_Count[4];
		ELSIF In_Hour_Code=6
			THEN
				Running_Target_CountPrevHourTotal:= Shift_Report[0].Expected_Count[1]+
													Shift_Report[0].Expected_Count[2]+
													Shift_Report[0].Expected_Count[3]+
													Shift_Report[0].Expected_Count[4]+
													Shift_Report[0].Expected_Count[5];
		ELSIF In_Hour_Code=7
			THEN
				Running_Target_CountPrevHourTotal:= Shift_Report[0].Expected_Count[1]+
													Shift_Report[0].Expected_Count[2]+
													Shift_Report[0].Expected_Count[3]+
													Shift_Report[0].Expected_Count[4]+
													Shift_Report[0].Expected_Count[5]+
													Shift_Report[0].Expected_Count[6];
		ELSIF In_Hour_Code=8
			THEN
				Running_Target_CountPrevHourTotal:= Shift_Report[0].Expected_Count[1]+
													Shift_Report[0].Expected_Count[2]+
													Shift_Report[0].Expected_Count[3]+
													Shift_Report[0].Expected_Count[4]+
													Shift_Report[0].Expected_Count[5]+
													Shift_Report[0].Expected_Count[6]+
													Shift_Report[0].Expected_Count[7];
		ELSIF In_Hour_Code=9
			THEN
				Running_Target_CountPrevHourTotal:= Shift_Report[0].Expected_Count[1]+
													Shift_Report[0].Expected_Count[2]+
													Shift_Report[0].Expected_Count[3]+
													Shift_Report[0].Expected_Count[4]+
													Shift_Report[0].Expected_Count[5]+
													Shift_Report[0].Expected_Count[6]+
													Shift_Report[0].Expected_Count[7]+
													Shift_Report[0].Expected_Count[8];
		ELSIF In_Hour_Code=10
			THEN
				Running_Target_CountPrevHourTotal:= Shift_Report[0].Expected_Count[1]+
													Shift_Report[0].Expected_Count[2]+
													Shift_Report[0].Expected_Count[3]+
													Shift_Report[0].Expected_Count[4]+
													Shift_Report[0].Expected_Count[5]+
													Shift_Report[0].Expected_Count[6]+
													Shift_Report[0].Expected_Count[7]+
													Shift_Report[0].Expected_Count[8]+
													Shift_Report[0].Expected_Count[9];
		ELSIF In_Hour_Code=11
			THEN
				Running_Target_CountPrevHourTotal:= Shift_Report[0].Expected_Count[1]+
													Shift_Report[0].Expected_Count[2]+
													Shift_Report[0].Expected_Count[3]+
													Shift_Report[0].Expected_Count[4]+
													Shift_Report[0].Expected_Count[5]+
													Shift_Report[0].Expected_Count[6]+
													Shift_Report[0].Expected_Count[7]+
													Shift_Report[0].Expected_Count[8]+
													Shift_Report[0].Expected_Count[9]+
													Shift_Report[0].Expected_Count[10];
		ELSIF In_Hour_Code=12
			THEN
				Running_Target_CountPrevHourTotal:= Shift_Report[0].Expected_Count[1]+
													Shift_Report[0].Expected_Count[2]+
													Shift_Report[0].Expected_Count[3]+
													Shift_Report[0].Expected_Count[4]+
													Shift_Report[0].Expected_Count[5]+
													Shift_Report[0].Expected_Count[6]+
													Shift_Report[0].Expected_Count[7]+
													Shift_Report[0].Expected_Count[8]+
													Shift_Report[0].Expected_Count[9]+
													Shift_Report[0].Expected_Count[10]+
													Shift_Report[0].Expected_Count[11];
		END_IF;
	END_IF;

(*Reset At Shift Change*)
	IF Start_Shift_Trigger.Q
		THEN
		Running_Target_Count:= 0;
	END_IF;

(*----------------- Monitor Production Increments ----------------*)

	IF Prod_Inc AND (In_Day_Shift OR In_Aft_Shift OR In_Mid_Shift)
		THEN
		Production_Count:= Production_Count+1;
	END_IF;

	(*Reset At Shift Change*)
	IF Start_Shift_Trigger.Q
		THEN
		Production_Count:= 0;
	END_IF;

(*--------------- Generate Difference ---------------------------*)

	Running_Difference:= (Production_Count - Running_Target_Count);

(*------------------- Monitor Scrap Count -----------------------*)

	(*Increment Scrap Counter*)
	Scrap_Inc_Trigger.CLK:= Scrap_Inc;
	Scrap_Inc_Trigger();
	IF Scrap_Inc_Trigger.Q
		THEN
			Running_Scrap_Count:=Running_Scrap_Count+1;
	END_IF;
	(*Decrement Scrap Counter*)
	Scrap_Dec_Trigger.CLK:= Scrap_Dec;
	Scrap_Dec_Trigger();
	IF Scrap_Dec_Trigger.Q
		THEN
			Running_Scrap_Count:=Running_Scrap_Count-1;
	END_IF;

	(*Reset At Shift Change*)
	IF Start_Shift_Trigger.Q
		THEN
		Running_Scrap_Count:= 0;
	END_IF;

(*---------------- Monitor Machine Stopped By Fault Time and capture fault count -------------*)

		(*Capture previouslly occured fault time once fault ceases to exist*)
		Not_Faulted_Trigger.CLK:= NOT Machine_StoppedBy_Fault OR End_Shift_Trigger.Q;
		Not_Faulted_Trigger();
		IF Not_Faulted_Trigger.Q
			THEN
				Previous_Faulted_Time:= Total_Faulted_Time;
		END_IF;

		(*Capture Currently Occuring fault time*)
		Faulted_TMR.PT:= T#12H0M0S0MS;
		Faulted_TMR.IN:= (In_Day_Shift OR In_Aft_Shift OR In_Mid_Shift) AND
							Machine_StoppedBy_Fault AND NOT In_Break AND NOT In_Shift_Change
							AND NOT Start_Shift_Trigger.Q AND NOT End_Shift_Trigger.Q;
		Faulted_TMR();

		(*Display out total of previously captured faults + currently occuring faults for Total Time Faulted in real time*)
		Total_Faulted_Time:= Previous_Faulted_Time + Faulted_TMR.ET;

		(*Capture Fault event into a total count of faults for shift*)
		FaultCount_Inc_Trigger.CLK:= Faulted_TMR.IN;
		FaultCount_Inc_Trigger();
		IF FaultCount_Inc_Trigger.Q
			THEN
				Total_Fault_Count:= Total_Fault_Count+1;
		END_IF;


		(*Reset both fault times and fault event count at shift change*)
		IF Start_Shift_Trigger.Q
			THEN
				Previous_Faulted_Time:= T#0H0M0S;
				Total_Faulted_Time:= T#0H0M0S;
				Total_Fault_Count:= 0;
		END_IF;

(*------------------ Calculate Machine Running Time  ---------------*)

		Running_TotalBy_Expected:= UINT_TO_REAL(Running_Target_Count) * TIME_TO_REAL(Reference_Target_Time); (*In ms*)
		Running_TotalTime:= REAL_TO_TIME(Running_TotalBy_Expected) + Target_TMR.ET;

(*------------------ Calculate Machine Uptime -----------------------*)

	IF Running_TotalTime >=Total_Faulted_Time
		THEN
		Running_UpTime:= Running_TotalTime-Total_Faulted_Time;
	ELSE
		Running_UpTime:= INT_TO_TIME(0);
	END_IF;

(*------------------ Generate KPI - OEE ---------------------------------*)

	(*Calc Availability Eff. -  Percentage of time was the machine available when it was supposed to be*)
	IF TIME_TO_UINT(Running_TotalTime)>0
		THEN
			Running_AvailabilityEFF:= ((TIME_TO_REAL(Running_UpTime)/TIME_TO_REAL(Running_TotalTime))*100);
	ELSE
			Running_AvailabilityEFF:=0;
	END_IF;

	(*Calc Perfromance Eff. - Percentage of speed machine ran at vs expected (IE Operator performance)*)
	(*First calc virtual parts lost during faulted time*)
	IF TIME_TO_UINT(Reference_Target_Time)>0
		THEN
			PartsLost_From_Faults:= TIME_TO_REAL(Total_Faulted_Time)/TIME_TO_REAL(Reference_Target_Time);
	ELSE
			PartsLost_From_Faults:= 0;
	END_IF;
	(*Then calc performance*)
	IF Running_Target_Count>=1 AND (UINT_TO_REAL(Running_Target_Count)>=PartsLost_From_Faults) AND NOT Start_Shift_Trigger.Q
		THEN
			Running_PerformanceEFF:= (((UINT_TO_REAL(Production_Count)+PartsLost_From_Faults) /
										UINT_TO_REAL(Running_Target_Count)) *100);
	ELSIF Running_Target_Count>=1 AND (UINT_TO_REAL(Running_Target_Count)<PartsLost_From_Faults) AND NOT Start_Shift_Trigger.Q
		THEN
			Running_PerformanceEFF:= 100;

	ELSIF Start_Shift_Trigger.Q
		THEN
			Running_PerformanceEFF:=0;
	END_IF;

	(*Calc Quality Eff*)
	IF Production_Count>0
		THEN
			Running_QualityEFF:= ((UINT_TO_REAL(Production_Count) - UINT_TO_REAL(Running_Scrap_Count))/
								UINT_TO_REAL(Production_Count)*100);
	ELSE
		Running_QualityEFF:=100;
	END_IF;

	(*Calc KPI OEE*)

		Running_OEE:= (Running_AvailabilityEFF * Running_PerformanceEFF * Running_QualityEFF) / 10000;

(* ------------------ Generate Report Status ------------------*)

	IF  FB_OK AND (In_Day_Shift OR In_Aft_Shift OR In_Mid_Shift)
		AND NOT In_Shift_Change AND NOT End_Shift_Trigger.CLK
		THEN
		(*In Shift messages*)
		IF In_Day_Shift
			THEN
			IF Faulted_TMR.IN
				THEN
					Status:= CONCAT('Day Shift, Faulted, Hour #', UINT_TO_STRING(In_Hour_Code));
			ELSIF In_Break
				THEN
					Status:= CONCAT('Day Shift, In Break, Hour #', UINT_TO_STRING(In_Hour_Code));
			ELSE
				Status:= CONCAT('Day Shift, Running, Hour #', UINT_TO_STRING(In_Hour_Code));
			END_IF;

		ELSIF In_Aft_Shift
			THEN
			IF Faulted_TMR.IN
				THEN
					Status:= CONCAT('Afternoon Shift, Faulted, Hour #', UINT_TO_STRING(In_Hour_Code));
			ELSIF In_Break
				THEN
					Status:= CONCAT('Afternoon Shift, In Break, Hour #', UINT_TO_STRING(In_Hour_Code));
			ELSE
				Status:= CONCAT('Afternoon Shift, Running, Hour #', UINT_TO_STRING(In_Hour_Code));
			END_IF;

		ELSIF In_Mid_Shift
			THEN
			IF Faulted_TMR.IN
				THEN
					Status:= CONCAT('Midnight Shift, Faulted, Hour #', UINT_TO_STRING(In_Hour_Code));
			ELSIF In_Break
				THEN
					Status:= CONCAT('Midnight Shift, In Break, Hour #', UINT_TO_STRING(In_Hour_Code));
			ELSE
				Status:= CONCAT('Midnight Shift, Running, Hour #', UINT_TO_STRING(In_Hour_Code));
			END_IF;

		END_IF;

	(*Paused for Shift Change*)
	ELSIF In_Shift_Change AND NOT End_Shift_Trigger.CLK
		THEN
		Status:= 'Paused for Shift Change';

	ELSIF End_Shift_Trigger.CLK
		THEN
		Status:= 'Ending Shift';

	(*Not in shift message*)
	ELSIF FB_OK AND NOT In_Day_Shift AND NOT In_Aft_Shift AND NOT In_Mid_Shift
		THEN
		Status:= 'Not in a Shift';

	(*Config Fault Messages*)
	ELSIF NOT FB_OK
		THEN
		IF NOT Day_Shift_ConfigOK
			THEN
			Status:= 'Day Shift Configuration Fault';
		ELSIF NOT Aft_Shift_ConfigOK
			THEN
			Status:= 'Afternoon Shift Configuration Fault';
		ELSIF NOT Mid_Shift_ConfigOK
			THEN
			Status:= 'Midnight Shift Configuration Fault';
		END_IF;

	ELSE
			Status:= 'unknown status, see FW dev.';
	END_IF;

(* --------------- Generate Shift Report -------------------------*)

	(*Generate Auto Shift Report*)
	IF (In_Day_Shift OR In_Aft_Shift OR In_Mid_Shift) AND Report_In_Auto
		THEN

			(*Generate Empty Data Area At Start Of Shift and Stamp With Time and Date*)
			IF Start_Shift_Trigger.Q AND NOT End_Shift_Trigger.Q
				THEN
					(*Set Time and Date Stamps*)
					Shift_Report[0].Start_Shift_TimeDate:= Reference_TimeDate;
					(*Blank Shift End Time*)
					Shift_Report[0].End_Shift_TimeDate.wYear:=0;
					Shift_Report[0].End_Shift_TimeDate.wMonth:=0;
					Shift_Report[0].End_Shift_TimeDate.wDay:=0;
					Shift_Report[0].End_Shift_TimeDate.wDayOfWeek:=0;
					Shift_Report[0].End_Shift_TimeDate.wHour:=0;
					Shift_Report[0].End_Shift_TimeDate.wMinute:=0;
					Shift_Report[0].End_Shift_TimeDate.wSecond:=0;
					Shift_Report[0].End_Shift_TimeDate.wMilliseconds:=0;
					(*Blank Shift Durations*)
					Shift_Report[0].Gross_Shift_Duration:= 0;
					Shift_Report[0].Net_Shift_Duration:= 0;
					(*Blank Machine and Common Data*)
					Shift_Report[0].Machine_Serial:= '';
					Shift_Report[0].Machine_Common_Name:= '';
					Shift_Report[0].Operator_ID:= 0;
					Shift_Report[0].Target_Cycle_Time:=T#0H0M0S;
					Shift_Report[0].Prod_Static_Target:=0;
					Shift_Report[0].Prod_Running_Target:=0;
					Shift_Report[0].Prod_Count_Total:=0;
					Shift_Report[0].Prod_Count_Scrap:=0;
					Shift_Report[0].Prod_Difference:=0;
					Shift_Report[0].Prod_Availability:=0;
					Shift_Report[0].Prod_Performance:=0;
					Shift_Report[0].Prod_Quality:=0;
					Shift_Report[0].Prod_Running_OEE:=0;
					Shift_Report[0].Prod_AvgFinal_PPH:=0;
					Shift_Report[0].Total_Fault_Time:=T#0H0M0S;
					Shift_Report[0].Total_Fault_Count:= 0;
					Shift_Report[0].Running_Up_Time:= T#0H0M0S;
					Shift_Report[0].Status:='';
					(*Blank Hourly Shift Data*)
					Shift_Report[0].Hour_Count[1]:=0;
					Shift_Report[0].Hour_Count[2]:=0;
					Shift_Report[0].Hour_Count[3]:=0;
					Shift_Report[0].Hour_Count[4]:=0;
					Shift_Report[0].Hour_Count[5]:=0;
					Shift_Report[0].Hour_Count[6]:=0;
					Shift_Report[0].Hour_Count[7]:=0;
					Shift_Report[0].Hour_Count[8]:=0;
					Shift_Report[0].Hour_Count[9]:=0;
					Shift_Report[0].Hour_Count[10]:=0;
					Shift_Report[0].Hour_Count[11]:=0;
					Shift_Report[0].Hour_Count[12]:=0;
					Shift_Report[0].Total_Count[1]:=0;
					Shift_Report[0].Total_Count[2]:=0;
					Shift_Report[0].Total_Count[3]:=0;
					Shift_Report[0].Total_Count[4]:=0;
					Shift_Report[0].Total_Count[5]:=0;
					Shift_Report[0].Total_Count[6]:=0;
					Shift_Report[0].Total_Count[7]:=0;
					Shift_Report[0].Total_Count[8]:=0;
					Shift_Report[0].Total_Count[9]:=0;
					Shift_Report[0].Total_Count[10]:=0;
					Shift_Report[0].Total_Count[11]:=0;
					Shift_Report[0].Total_Count[12]:=0;
					Shift_Report[0].Expected_Count[1]:=0;
					Shift_Report[0].Expected_Count[2]:=0;
					Shift_Report[0].Expected_Count[3]:=0;
					Shift_Report[0].Expected_Count[4]:=0;
					Shift_Report[0].Expected_Count[5]:=0;
					Shift_Report[0].Expected_Count[6]:=0;
					Shift_Report[0].Expected_Count[7]:=0;
					Shift_Report[0].Expected_Count[8]:=0;
					Shift_Report[0].Expected_Count[9]:=0;
					Shift_Report[0].Expected_Count[10]:=0;
					Shift_Report[0].Expected_Count[11]:=0;
					Shift_Report[0].Expected_Count[12]:=0;
			(*Build Current Report*)
			ELSIF NOT Start_Shift_Trigger.Q AND NOT End_Shift_Trigger.Q
				THEN
							(*Set Machine and Operator Data and Target CT*)
							Shift_Report[0].Machine_Serial:= Machine_Serial;
							Shift_Report[0].Machine_Common_Name:= Machine_Common_Name;
							Shift_Report[0].Operator_ID:= Operator_ID;
							Shift_Report[0].Target_Cycle_Time:= Reference_Target_Time;
							(*Capture shift configuration data*)
							Shift_Report[0].ProdConfig_Common.Break_Count:= Config_Break_Count;
							Shift_Report[0].ProdConfig_Common.Shift_Enables:= Config_Shift_Enables;
							Shift_Report[0].ProdConfig_Common.Config_Option_Flags.0:= Enable_InShift_Change;
								IF In_Day_Shift
									THEN
									Shift_Report[0].ProdConfig_Times:= FUN_GTAC_TODtoUDINT(Config_Day_TOD);
								ELSIF In_Aft_Shift
									THEN
									Shift_Report[0].ProdConfig_Times:= FUN_GTAC_TODtoUDINT(Config_Aft_TOD);
								ELSIF In_Mid_Shift
									THEN
									Shift_Report[0].ProdConfig_Times:= FUN_GTAC_TODtoUDINT(Config_Mid_TOD);
								END_IF;
							(*Set Shift Durations*)
							Shift_Report[0].Gross_Shift_Duration:= Gross_Shift_Duration;
							Shift_Report[0].Net_Shift_Duration:= Net_Shift_Duration;
							(*Transfer Common Data*)
							Shift_Report[0].Prod_Static_Target:= Static_Target;
							Shift_Report[0].Prod_Running_Target:= Running_Target_Count;
							Shift_Report[0].Prod_Count_Total:= Production_Count;
							Shift_Report[0].Prod_Count_Scrap:=Running_Scrap_Count;
							Shift_Report[0].Prod_Difference:= Running_Difference;
							Shift_Report[0].Prod_Availability:= Running_AvailabilityEFF;
							Shift_Report[0].Prod_Performance:= Running_PerformanceEFF;
							Shift_Report[0].Prod_Quality:= Running_QualityEFF;
							Shift_Report[0].Prod_Running_OEE:= Running_OEE;
							Shift_Report[0].Total_Fault_Time:=Total_Faulted_Time;
							Shift_Report[0].Total_Fault_Count:= Total_Fault_Count;
							Shift_Report[0].Running_Up_Time:= Running_UpTime;
							Shift_Report[0].Status:= Status;
							(*Transfer Hourly Data*)
							Shift_Report[0].Total_Count[In_Hour_Code]:= Shift_Report[0].Prod_Count_Total;
							IF In_Hour_Code=1
								THEN
									(*Calc Hourly Production*)
									Shift_Report[0].Hour_Count[In_Hour_Code]:= Shift_Report[0].Prod_Count_Total;
									(*Calc Hourly Expected*)
									Shift_Report[0].Expected_Count[In_Hour_Code]:= Shift_Report[0].Prod_Running_Target;
							ELSIF In_Hour_Code>=2
								THEN
									(*Calc Hourly Production*)
									Shift_Report[0].Hour_Count[In_Hour_Code]:=
										Shift_Report[0].Prod_Count_Total - Shift_Report[0].Total_Count[In_Hour_Code - 1];
									(*Calc Hourly Expected*)
									Shift_Report[0].Expected_Count[In_Hour_Code]:=
										Shift_Report[0].Prod_Running_Target - Running_Target_CountPrevHourTotal;
							END_IF;
			(*Finazlize Report At End Of Shift*)
			ELSIF End_Shift_Trigger.Q
				THEN
					(*Take Snap Shot of End of Shift Time*)
					Shift_Report[0].End_Shift_TimeDate:= Reference_TimeDate;
					(*Mark Report Status as completed*)
					Shift_Report[0].Status:= 'Shift Completed';
					(*Calc Totals etc*)
					IF Net_Shift_Duration>0
						THEN
						Shift_Report[0].Prod_AvgFinal_PPH:= UINT_TO_REAL(Shift_Report[0].Prod_Count_Total) / Net_Shift_Duration;
					ELSE
						Shift_Report[0].Prod_AvgFinal_PPH:= Shift_Report[0].Prod_Count_Total/8; (*Default*)
					END_IF;
					IF In_Shift_Code >0 AND In_Shift_Code <=3
						THEN
						Shift_Report[In_Shift_Code]:=Shift_Report[0];	(*At End Of Shift, Capture Current Shift Data to Current Shift History Area*)
					END_IF;
			END_IF;
	ELSE (*Not in Any Shift then Allow Status through for indication of "Not in Shift"*)
		Shift_Report[0].Status:= Status;
	END_IF;(*End Of Auto Report Generator*)

(*------------------------------------------------------------------------- Shift Report Override Mode Code -------------------------------------------------------*)
(*!!!!!!!!!!!For Future Development!!!!!!!!!!!!*)

ACTION ShiftConfigs_TOD_To_OTSTRUCT:
	(*Day Shift*)
	Config_Day.Shift_StartTime:= FUN_GTAC_TODtoOTSTRUCT(Config_Day_TOD.Shift_StartTime);
		Config_Day.Break1_StartTime:= FUN_GTAC_TODtoOTSTRUCT(Config_Day_TOD.Break1_StartTime);
		Config_Day.Break1_EndTime:= FUN_GTAC_TODtoOTSTRUCT(Config_Day_TOD.Break1_EndTime);
		Config_Day.Break2_StartTime:= FUN_GTAC_TODtoOTSTRUCT(Config_Day_TOD.Break2_StartTime);
		Config_Day.Break2_EndTime:= FUN_GTAC_TODtoOTSTRUCT(Config_Day_TOD.Break2_EndTime);
		Config_Day.Break3_StartTime:= FUN_GTAC_TODtoOTSTRUCT(Config_Day_TOD.Break3_StartTime);
		Config_Day.Break3_EndTime:= FUN_GTAC_TODtoOTSTRUCT(Config_Day_TOD.Break3_EndTime);
	Config_Day.Shift_EndTime:= FUN_GTAC_TODtoOTSTRUCT(Config_Day_TOD.Shift_EndTime);


	(*Afternoon Shift*)
	Config_Aft.Shift_StartTime:= FUN_GTAC_TODtoOTSTRUCT(Config_Aft_TOD.Shift_StartTime);
		Config_Aft.Break1_StartTime:= FUN_GTAC_TODtoOTSTRUCT(Config_Aft_TOD.Break1_StartTime);
		Config_Aft.Break1_EndTime:= FUN_GTAC_TODtoOTSTRUCT(Config_Aft_TOD.Break1_EndTime);
		Config_Aft.Break2_StartTime:= FUN_GTAC_TODtoOTSTRUCT(Config_Aft_TOD.Break2_StartTime);
		Config_Aft.Break2_EndTime:= FUN_GTAC_TODtoOTSTRUCT(Config_Aft_TOD.Break2_EndTime);
		Config_Aft.Break3_StartTime:= FUN_GTAC_TODtoOTSTRUCT(Config_Aft_TOD.Break3_StartTime);
		Config_Aft.Break3_EndTime:= FUN_GTAC_TODtoOTSTRUCT(Config_Aft_TOD.Break3_EndTime);
	Config_Aft.Shift_EndTime:= FUN_GTAC_TODtoOTSTRUCT(Config_Aft_TOD.Shift_EndTime);


	(*Midnight Shift*)
	Config_Mid.Shift_StartTime:= FUN_GTAC_TODtoOTSTRUCT(Config_Mid_TOD.Shift_StartTime);
		Config_Mid.Break1_StartTime:= FUN_GTAC_TODtoOTSTRUCT(Config_Mid_TOD.Break1_StartTime);
		Config_Mid.Break1_EndTime:= FUN_GTAC_TODtoOTSTRUCT(Config_Mid_TOD.Break1_EndTime);
		Config_Mid.Break2_StartTime:= FUN_GTAC_TODtoOTSTRUCT(Config_Mid_TOD.Break2_StartTime);
		Config_Mid.Break2_EndTime:= FUN_GTAC_TODtoOTSTRUCT(Config_Mid_TOD.Break2_EndTime);
		Config_Mid.Break3_StartTime:= FUN_GTAC_TODtoOTSTRUCT(Config_Mid_TOD.Break3_StartTime);
		Config_Mid.Break3_EndTime:= FUN_GTAC_TODtoOTSTRUCT(Config_Mid_TOD.Break3_EndTime);
	Config_Mid.Shift_EndTime:= FUN_GTAC_TODtoOTSTRUCT(Config_Mid_TOD.Shift_EndTime);
END_ACTION

END_FUNCTION_BLOCK

// ---- POUs/FUNs/FUN_GTAC_TIMESTRUCTtoTOD.TcPOU
(*Take Individual time elements of a TIMESTRUCT and create a TOD type return
	author: Brent Lekx-Toniolo Of Sodecia GTAC
	date: May 2016
	version 1.0
		- initial concept


	Last Edit: 27-May-2016, blt
*)

FUNCTION FUN_GTAC_TIMESTRUCTtoTOD : TOD
VAR_INPUT
	TIMESTRUCT: TIMESTRUCT;

END_VAR
VAR
	Hours_as_MS: UDINT;
	Minutes_as_MS: UDINT;
	Seconds_as_MS: UDINT;
	Milliseconds_as_MS: UDINT;
END_VAR

(*Calculate Millsecond Value of each OTSTRUCT Element*)

	Hours_as_MS:= TIMESTRUCT.wHour * 3600000;
	Minutes_as_MS:= TIMESTRUCT.wMinute * 60000;
	Seconds_as_MS:= TIMESTRUCT.wSecond * 1000;
	Milliseconds_as_MS:= TIMESTRUCT.wMilliseconds;

(*Return Total Value in Milliseconds, this is TOD*)

	FUN_GTAC_TIMESTRUCTtoTOD:= UDINT_TO_TOD(Hours_As_MS + Minutes_As_MS + Seconds_As_MS + Milliseconds_As_MS);

END_FUNCTION

// ---- POUs/FUNs/FUN_GTAC_ReturnGrossShiftDuration.TcPOU
(*Uses Shift Configuration Structure and calculates total Gross duration of shift time (in hours)
	original author: Brent Lekx-Toniolo of Fort Wisers / OoR Tech

----------------------------------------------------------------------------------------------------------------------
REVISION NOTES: 
	Date: Jan 22, 2020:
	- initial concept, blt
	Date: October 25, 2022
	- Added type conversaion to supress build warning, b.lekx-toniolo

------------------------------------------------------------------------------------------------------------------------	

*)

FUNCTION FUN_GTAC_ReturnGrossShiftDuration: REAL
VAR_INPUT
	Shift_Config_TOD: udt_Generic_ShiftConfigTOD_20160527;
END_VAR
VAR

	Gross_Duration_Milliseconds: REAL;
	Gross_Duration_Hours: REAL;


END_VAR

(*Calcuate Gross Shift Duration in milliseconds*)
	IF Shift_Config_TOD.Shift_EndTime > Shift_Config_TOD.Shift_StartTime
		THEN
		Gross_Duration_Milliseconds:= UDINT_TO_REAL (TOD_TO_UDINT(Shift_Config_TOD.Shift_EndTime) - TOD_TO_UDINT(Shift_Config_TOD.Shift_StartTime));
	ELSIF Shift_Config_TOD.Shift_EndTime < Shift_Config_TOD.Shift_StartTime
		THEN
		Gross_Duration_Milliseconds:= UDINT_TO_REAL(( 86400000 - TOD_TO_UDINT(Shift_Config_TOD.Shift_StartTime)) + TOD_TO_UDINT(Shift_Config_TOD.Shift_EndTime));
	END_IF;

(*Calcualte Milliseconds to Hours*)
	Gross_Duration_Hours:= Gross_Duration_Milliseconds / UDINT_TO_REAL((60*60*1000));


(*Finally, Return Value, in hours*)
	FUN_GTAC_ReturnGrossShiftDuration:= Gross_Duration_Hours;

END_FUNCTION

// ---- POUs/FUNs/FUN_GTAC_ReturnNetShiftDuration.TcPOU
(*Uses Shift Configuration Structure and calculates total Net duration of shift time (in hours)
	original author: Brent Lekx-Toniolo Of Sodecia GTAC

----------------------------------------------------------------------------------------------------------------------
REVISION NOTES: 
	Date: May 19, 2016:
	- initial concept, blt
	Date: Jan 22, 2020:
	- added in shift enables during production code updates, blt
	- changed all calcs and interface to remove the need of OTSTRUCT type data, blt
	Date: October 25, 2022
	- Added type conversaion to supress build warning, b.lekx-toniolo


------------------------------------------------------------------------------------------------------------------------	

*)

FUNCTION FUN_GTAC_ReturnNetShiftDuration: REAL
VAR_INPUT
	Shift_Config_TOD: udt_Generic_ShiftConfigTOD_20160527;
	Break_Count: UINT;
END_VAR
VAR
	Gross_Duration_Milliseconds: REAL;
	Break1_Duration_Milliseconds: REAL;
	Break2_Duration_Milliseconds: REAL;
	Break3_Duration_Milliseconds: REAL;

	Net_Duration_Milliseconds: REAL;
	Net_Duration_Hours: REAL;
END_VAR

(*Calcuate Gross Shift Duration in milliseconds*)
	IF Shift_Config_TOD.Shift_EndTime > Shift_Config_TOD.Shift_StartTime
		THEN
		Gross_Duration_Milliseconds:= UDINT_TO_REAL(TOD_TO_UDINT(Shift_Config_TOD.Shift_EndTime) - TOD_TO_UDINT(Shift_Config_TOD.Shift_StartTime));
	ELSIF Shift_Config_TOD.Shift_EndTime < Shift_Config_TOD.Shift_StartTime
		THEN
		Gross_Duration_Milliseconds:= UDINT_TO_REAL(( 86400000 - TOD_TO_UDINT(Shift_Config_TOD.Shift_StartTime)) + TOD_TO_UDINT(Shift_Config_TOD.Shift_EndTime));
	END_IF;


(*Calcuate Break1 Duration*)
	IF (Break_Count >=1)
		THEN
		(*Calc break duration*)
		IF Shift_Config_TOD.Break1_EndTime > Shift_Config_TOD.Break1_StartTime
			THEN
		Break1_Duration_Milliseconds:= UDINT_TO_REAL(TOD_TO_UDINT(Shift_Config_TOD.Break1_EndTime) - TOD_TO_UDINT(Shift_Config_TOD.Break1_StartTime));
		ELSIF Shift_Config_TOD.Break1_EndTime < Shift_Config_TOD.Break1_StartTime
			THEN
		Break1_Duration_Milliseconds:= UDINT_TO_REAL(( 86400000 - TOD_TO_UDINT(Shift_Config_TOD.Break1_StartTime)) + TOD_TO_UDINT(Shift_Config_TOD.Break1_EndTime));
		END_IF;
	ELSE
	(*If break is disable, blank duration*)
	Break1_Duration_Milliseconds:= 0;
	END_IF;

(*Calcuate Break2 Duration*)
	IF (Break_Count >=2)
		THEN
		(*Calc break duration*)
		IF Shift_Config_TOD.Break2_EndTime > Shift_Config_TOD.Break2_StartTime
			THEN
		Break2_Duration_Milliseconds:= UDINT_TO_REAL(TOD_TO_UDINT(Shift_Config_TOD.Break2_EndTime) - TOD_TO_UDINT(Shift_Config_TOD.Break2_StartTime));
		ELSIF Shift_Config_TOD.Break2_EndTime < Shift_Config_TOD.Break2_StartTime
			THEN
		Break2_Duration_Milliseconds:= UDINT_TO_REAL(( 86400000 - TOD_TO_UDINT(Shift_Config_TOD.Break2_StartTime)) + TOD_TO_UDINT(Shift_Config_TOD.Break2_EndTime));
		END_IF;
	ELSE
	(*If break is disable, blank duration*)
	Break2_Duration_Milliseconds:= 0;
	END_IF;

(*Calcuate Break3 Duration*)
	IF (Break_Count >=3)
		THEN
		(*Calc break duration*)
		IF Shift_Config_TOD.Break3_EndTime > Shift_Config_TOD.Break3_StartTime
			THEN
		Break3_Duration_Milliseconds:= UDINT_TO_REAL(TOD_TO_UDINT(Shift_Config_TOD.Break3_EndTime) - TOD_TO_UDINT(Shift_Config_TOD.Break3_StartTime));
		ELSIF Shift_Config_TOD.Break3_EndTime < Shift_Config_TOD.Break3_StartTime
			THEN
		Break3_Duration_Milliseconds:= UDINT_TO_REAL(( 86400000 - TOD_TO_UDINT(Shift_Config_TOD.Break3_StartTime)) + TOD_TO_UDINT(Shift_Config_TOD.Break3_EndTime));
		END_IF;
	ELSE
	(*If break is disable, blank duration*)
	Break3_Duration_Milliseconds:= 0;
	END_IF;

(*----------------------------------------------------------------------------------------- Generate Function Output ----------------------------------------------------------------*)
(*Remove break durations from gross duration*)
	Net_Duration_Milliseconds:= Gross_Duration_Milliseconds - Break1_Duration_Milliseconds - Break2_Duration_Milliseconds - Break3_Duration_Milliseconds;

(*Calcualte Milliseconds to Hours*)
	Net_Duration_Hours:= Net_Duration_Milliseconds / UDINT_TO_REAL((60*60*1000));

(*Finally, Return Value*)
	FUN_GTAC_ReturnNetShiftDuration:= Net_Duration_Hours;

END_FUNCTION

